Yaskawa INFORM job: X2_8A-21A(90,0)_REV_O.JBI

/JOB
//NAME X2_8A-21A(90,0)_REV_O
///FOLDERNAME X2
//POS
///NPOS 1933,1933,1933,50,0,0
///TOOL 0
///POSTYPE PULSE
///PULSE
C00000=-12667,-135547,-130714,31270,45596,0
C00001=-9315,-159766,-119262,-3212,6219,55552
C00002=-157761,-135547,-130714,31270,45596,-69143
C00003=-154472,-113934,-104337,41712,51336,-70449
C00004=-149832,-108771,-100172,39130,49259,-68869
C00005=-148058,-106656,-98467,38074,48499,-68236
C00006=-148062,-106275,-96666,38578,47777,-68578
C00007=-148058,-106656,-98467,38074,48499,-68236
C00008=-147997,-106381,-96958,38469,47847,-68508
C00009=-145894,-104035,-96109,36815,47477,-67498
C00010=-147997,-106381,-96958,38469,47847,-68508
C00011=-154410,-113635,-102825,42095,50721,-70729
C00012=-154342,-120637,-107041,25827,48602,-38771
C00013=-150292,-111683,-102360,22573,48994,-36710
C00014=-148798,-108210,-100464,21373,49171,-35962
C00015=-146664,-105787,-99597,19708,49308,-34937
C00016=-146949,-106220,-99797,19932,49282,-35074
C00017=-147721,-103636,-97533,20478,49410,-35405
C00018=-146949,-106220,-99797,19932,49282,-35074
C00019=-152261,-118724,-106469,24248,48548,-37770
C00020=-148295,-114597,-117137,-6490,60568,-69086
C00021=-147868,-109631,-111600,-6790,59752,-68875
C00022=-117093,-120499,-115228,-23648,62285,-57221
C00023=-113886,-102168,-107256,-24278,67338,-57062
C00024=-113886,-102375,-106001,-24426,66534,-56885
C00025=-113886,-102359,-106115,-24413,66607,-56901
C00026=-113886,-102359,-106115,-24413,66607,-56901
C00027=-114646,-97769,-104385,-23859,67577,-57404
C00028=-114475,-101992,-107821,-23944,67574,-57337
C00029=-147704,-107727,-109395,-6911,59390,-68790
C00030=-147708,-107860,-107783,-6984,58336,-68724
C00031=-147704,-107727,-109395,-6911,59390,-68790
C00032=-147723,-107760,-107968,-6963,58499,-68740
C00033=-147306,-102596,-106094,-7098,60024,-68678
C00034=-147723,-107760,-107968,-6963,58499,-68740
C00035=-148315,-114751,-115749,-6537,59639,-69038
C00036=-148355,-114889,-117236,-6461,60467,-69101
C00037=-147925,-109892,-111692,-6763,59663,-68890
C00038=-147761,-107977,-109485,-6884,59305,-68805
C00039=-147764,-108104,-107870,-6957,58254,-68739
C00040=-147777,-108153,-108078,-6942,58354,-68751
C00041=-147358,-102980,-106206,-7078,59886,-68688
C00042=-147777,-108153,-108078,-6942,58354,-68751
C00043=-148373,-115211,-115873,-6515,59468,-69049
C00044=-147696,-122269,-111871,-35505,39043,-51945
C00045=-147690,-118447,-100224,-39719,34874,-49579
C00046=-148491,-109409,-94254,-38171,35277,-50420
C00047=-148787,-105724,-91002,-38010,35060,-50504
C00048=-148789,-105382,-89977,-38411,34697,-50285
C00049=-149058,-101689,-89016,-37046,35623,-51030
C00050=-149145,-100783,-88679,-36755,35795,-51189
C00051=-149058,-101689,-89016,-37046,35623,-51030
C00052=-145777,-99657,-88811,-39022,37803,-49998
C00053=-148139,-100407,-89095,-37251,36591,-50936
C00054=-145777,-99657,-88811,-39022,37803,-49998
C00055=-147690,-118447,-100224,-39719,34874,-49579
C00056=-128033,-128545,-103748,-39689,32513,-43973
C00057=-128383,-118409,-97778,-37905,33566,-44930
C00058=-128511,-114277,-94563,-37658,33626,-45064
C00059=-128512,-113804,-93446,-38069,33271,-44843
C00060=-129119,-111006,-93029,-36452,33958,-45715
C00061=-129434,-109852,-92636,-35862,34111,-46033
C00062=-128358,-113721,-93936,-37885,33613,-44941
C00063=-176216,-70111,-78093,55162,70856,-80763
C00064=-174311,-70781,-78417,54616,69674,-80426
C00065=-176216,-70111,-78093,55162,70856,-80763
C00066=-181747,-69996,-81392,56304,75271,-81045
C00067=-178033,-77165,-93769,42680,75059,-77098
C00068=-164745,-109340,-116699,-3009,62053,-68278
C00069=-145851,-112599,-102075,-47717,41998,-56322
C00070=-148044,-104803,-96379,-45883,41204,-57334
C00071=-148864,-101708,-93474,-45490,40644,-57533
C00072=-148866,-101457,-92299,-45986,40221,-57239
C00073=-148863,-101834,-94104,-45225,40876,-57690
C00074=-145127,-99228,-91361,-47944,42572,-56214
C00075=-147466,-100038,-91670,-46636,41186,-56907
C00076=-145127,-99228,-91361,-47944,42572,-56214
C00077=-146129,-107372,-95667,-48598,40993,-55782
C00078=-148216,-109089,-93488,-49289,38371,-55335
C00079=-148344,-107837,-93052,-48851,38553,-55585
C00080=-147906,-112054,-94498,-50363,37947,-54724
C00081=-145851,-112599,-102075,-47717,41998,-56322
C00082=-158250,-140903,-124067,-47621,67451,-49320
C00083=-161740,-133075,-117656,-46661,65672,-50232
C00084=-162335,-130592,-114553,-46699,64919,-50156
C00085=-162276,-129951,-113381,-46845,64676,-49998
C00086=-160420,-132544,-115533,-47350,65644,-49520
C00087=-135901,-74424,-73697,-74364,100921,-31256
C00088=-137788,-75503,-74147,-74218,99532,-31324
C00089=-138769,-76027,-74362,-74146,98812,-31363
C00090=-135901,-74424,-73697,-74364,100921,-31256
C00091=-149282,-147643,-98518,-79858,51263,-26133
C00092=-149394,-146891,-98381,-79629,51249,-26315
C00093=-148448,-152811,-99407,-81432,51428,-24854
C00094=-139735,-166147,-105854,-82069,56849,-22658
C00095=-180438,-97574,-115199,-33764,102267,52414
C00096=-189965,-108899,-115705,-31971,94091,51156
C00097=-190633,-110068,-115194,-31831,93066,51189
C00098=-190637,-110288,-114404,-31804,92551,51332
C00099=-190629,-109833,-115910,-31859,93547,51055
C00100=-186867,-102382,-113240,-32521,96788,51574
C00101=-187005,-102964,-110979,-32373,95300,51952
C00102=-188888,-106610,-112304,-32065,93703,51681
C00103=-187005,-102964,-110979,-32373,95300,51952
C00104=-188021,-107681,-112675,-32159,93748,52003
C00105=-189590,-103281,-111094,-32025,94271,51250
C00106=-188021,-107681,-112675,-32159,93748,52003
C00107=-180438,-97574,-115199,-33764,102267,52414
C00108=-185735,-83978,-109774,-33564,103394,50026
C00109=-199988,-77820,-108712,11582,98175,-38155
C00110=-204749,-56978,-92496,29836,109182,-47433
C00111=-202460,-56662,-91339,29422,107990,-46925
C00112=-201413,-57385,-91726,29256,107546,-46663
C00113=-201611,-57041,-91542,29296,107663,-46703
C00114=-201611,-58240,-90431,29070,106521,-47008
C00115=-203359,-50274,-87822,29763,109247,-46906
C00116=-195470,-25798,-72981,29209,109868,-43903
C00117=-195013,-27562,-73704,29036,109327,-43888
C00118=-194283,-28250,-74172,28893,109053,-43704
C00119=-194480,-28066,-74047,28932,109127,-43754
C00120=-194480,-29296,-73135,28708,108075,-44034
C00121=-195605,-24849,-71507,29147,109538,-44038
C00122=-191110,-5546,-57842,28597,109561,-42465
C00123=-192519,-3768,-54500,33008,111368,-41387
C00124=-191992,-5303,-55742,32912,111174,-41254
C00125=-192059,-5108,-55586,32924,111198,-41271
C00126=-192059,-6294,-54683,32651,110210,-41583
C00127=-192882,-2296,-53893,33162,111810,-41382
C00128=-203365,-15491,-64400,34648,115083,-44256
C00129=-218411,-26661,-75493,58573,107247,-46176
C00130=-145332,-87800,-123084,4045,108310,15756
C00131=-109199,-104290,-129101,-21867,105305,43874
C00132=-112610,-115777,-129409,-14908,94573,36374
C00133=-117115,-112620,-124614,-14006,92529,35127
C00134=-122920,-112365,-123082,-12804,90828,33394
C00135=-122920,-112757,-122533,-12801,90299,33450
C00136=-122920,-112643,-122701,-12801,90458,33434
C00137=-123525,-106184,-120478,-12700,92275,33049
C00138=-122920,-112643,-122701,-12801,90458,33434
C00139=-99736,-107822,-114568,-33675,94477,38345
C00140=-104025,-110392,-115465,-33031,92199,37352
C00141=-122920,-112281,-123196,-12806,90936,33384
C00142=-119624,-116552,-128230,-13509,92325,34321
C00143=-118894,-118314,-126738,-16484,89836,32308
C00144=-120722,-107922,-120892,-16116,91165,31519
C00145=-120722,-108682,-119869,-16105,90184,31649
C00146=-120722,-108549,-120061,-16106,90363,31625
C00147=-121452,-100742,-117219,-15984,92406,31115
C00148=-121469,-105211,-119242,-15960,91389,31241
C00149=-101189,-106149,-119574,-19874,95347,37480
C00150=-117231,-121833,-124467,-22052,85463,28755
C00151=-122341,-114124,-118662,-20866,84531,27121
C00152=-123318,-113111,-117155,-20643,83910,26885
C00153=-123641,-113323,-116249,-20585,83205,26892
C00154=-123595,-112804,-116375,-20585,83540,26851
C00155=-123397,-106736,-114247,-20589,85286,26623
C00156=-123595,-112804,-116375,-20585,83540,26851
C00157=-116023,-114044,-115764,-22346,84523,29358
C00158=-117346,-116777,-115957,-22098,82979,29171
C00159=-118867,-116723,-116143,-21757,82713,28674
C00160=-116293,-116772,-115815,-22329,83179,29512
C00161=-117231,-121833,-124467,-22052,85463,28755
C00162=-154726,-134692,-133300,19029,79240,32627
C00163=-155157,-123239,-125350,19102,80279,32639
C00164=-157379,-119183,-122744,19707,81244,32017
C00165=-157379,-119362,-122195,19727,80834,31951
C00166=-157379,-119302,-122385,19720,80973,31974
C00167=-156300,-113680,-120537,19346,82380,32578
C00168=-157190,-118033,-122826,19626,81802,32175
C00169=-175737,-146891,-124533,43519,91428,21152
C00170=-174721,-145732,-123510,43532,90901,21397
C00171=-174058,-146263,-122600,43517,89962,21303
C00172=-174118,-146172,-122608,43517,90030,21304
C00173=-173980,-142501,-121319,43546,90763,21685
C00174=-177980,-148291,-122807,43386,91220,20037
C00175=-177422,-148804,-122388,43393,90560,20012
C00176=-177529,-148647,-122416,43390,90685,20016
C00177=-177298,-142861,-120187,43458,91752,20577
C00178=-177298,-144596,-123184,43505,92454,20876
C00179=-171479,-146654,-130538,32727,84182,23892
C00180=-166226,-153583,-132379,32233,80103,24817
C00181=-165373,-149023,-130107,32047,80585,25297
C00182=-165373,-148396,-128971,32075,80265,25206
C00183=-165373,-148499,-129154,32071,80317,25220
C00184=-163349,-139759,-126762,31573,82140,26540
C00185=-164602,-145870,-129723,31842,81480,25858
C00186=-94432,-122903,-125032,-9527,78085,47389
C00187=-94433,-123258,-123690,-9573,77094,47468
C00188=-95155,-123271,-123048,-9356,76614,47257
C00189=-95046,-123163,-123057,-9388,76686,47288
C00190=-95200,-117884,-121168,-9287,78202,47121
C00191=-91884,-123031,-122816,-10395,76986,48348
C00192=-93089,-124364,-122323,-10053,75863,48028
C00193=-92985,-124257,-122339,-10083,75941,48058
C00194=-93121,-120077,-120785,-9995,77098,47917
C00195=-92614,-123227,-123779,-10148,77379,48067
C00196=-142492,-148036,-131704,16940,70784,31434
C00197=-120610,-122471,-119242,-21572,81234,22537
C00198=-120610,-122484,-118172,-21604,80613,22649
C00199=-120610,-122391,-116483,-21658,79689,22817
C00200=-120610,-122419,-116833,-21647,79876,22783
C00201=-120610,-122423,-116832,-21647,79874,22783
C00202=-120610,-122419,-116833,-21647,79876,22783
C00203=-120610,-122416,-116761,-21649,79836,22790
C00204=-120610,-122436,-116768,-21650,79830,22791
C00205=-120610,-122416,-116761,-21649,79836,22790
C00206=-120611,-122370,-120508,-21535,82009,22397
C00207=-120500,-119354,-126515,-17332,87675,17755
C00208=-155157,-123239,-125350,19102,80279,32639
C00209=-157379,-119183,-122744,19707,81244,32017
C00210=-157379,-119362,-122195,19727,80834,31951
C00211=-157379,-119302,-122385,19720,80973,31974
C00212=-156300,-113680,-120537,19346,82380,32578
C00213=-157190,-118033,-122826,19626,81802,32175
C00214=-175737,-146891,-124533,43519,91428,21152
C00215=-174721,-145732,-123510,43532,90901,21397
C00216=-174058,-146263,-122600,43517,89962,21303
C00217=-174118,-146172,-122608,43517,90030,21304
C00218=-173980,-142501,-121319,43546,90763,21685
C00219=-177980,-148291,-122807,43386,91220,20037
C00220=-177422,-148804,-122388,43393,90560,20012
C00221=-177529,-148647,-122416,43390,90685,20016
C00222=-177298,-142861,-120187,43458,91752,20577
C00223=-177298,-144596,-123184,43505,92454,20876
C00224=-171479,-146654,-130538,32727,84182,23892
C00225=-166226,-153583,-132379,32233,80103,24817
C00226=-165373,-149023,-130107,32047,80585,25297
C00227=-165373,-148396,-128971,32075,80265,25206
C00228=-165373,-148499,-129154,32071,80317,25220
C00229=-163349,-139759,-126762,31573,82140,26540
C00230=-164602,-145870,-129723,31842,81480,25858
C00231=-94432,-122903,-125032,-9527,78085,47389
C00232=-94433,-123258,-123690,-9573,77094,47468
C00233=-95155,-123271,-123048,-9356,76614,47257
C00234=-95046,-123163,-123057,-9388,76686,47288
C00235=-95200,-117884,-121168,-9287,78202,47121
C00236=-91884,-123031,-122816,-10395,76986,48348
C00237=-93089,-124364,-122323,-10053,75863,48028
C00238=-92985,-124257,-122339,-10083,75941,48058
C00239=-93121,-120077,-120785,-9995,77098,47917
C00240=-92614,-123227,-123779,-10148,77379,48067
C00241=-120611,-118687,-129075,-3134,90000,4412
C00242=-148570,-103220,-123870,3202,94742,-4439
C00243=-148570,-107981,-119269,3182,89471,-4572
C00244=-127056,-134876,-126643,7466,81568,-11458
C00245=-127056,-134636,-125176,7474,80796,-11503
C00246=-127056,-134735,-125722,7473,81078,-11487
C00247=-126802,-126383,-123229,7383,83789,-11239
C00248=-127056,-134735,-125722,7473,81078,-11487
C00249=-152011,-114496,-114941,26277,90880,-36116
C00250=-148601,-117726,-116011,25806,88925,-35294
C00251=-149160,-116575,-119890,25935,91789,-34871
C00252=-149049,-114583,-124201,25964,95071,-34011
C00253=-120621,-113915,-131911,-13153,116790,34478
C00254=-136832,-143297,-133894,-19017,104291,40845
C00255=-187686,-122249,-118318,-34521,102174,42234
C00256=-187703,-122088,-115580,-34298,100833,42653
C00257=-187707,-122010,-114917,-34250,100525,42749
C00258=-187713,-121734,-113169,-34135,99743,42991
C00259=-187707,-122010,-114917,-34250,100525,42749
C00260=-187770,-121697,-112491,-32279,113674,44764
C00261=-187767,-121692,-112491,-32279,113678,44765
C00262=-187770,-121697,-112491,-32279,113674,44764
C00263=-187667,-121438,-112064,-34928,84963,41689
C00264=-187673,-121448,-112068,-34927,84958,41688
C00265=-187667,-121438,-112064,-34928,84963,41689
C00266=-187641,-121360,-124129,-34919,91154,39753
C00267=-178673,-119471,-127738,-23493,103847,53429
C00268=-198679,-138959,-135715,-16358,95506,85843
C00269=-190587,-123959,-122502,-31374,99801,86508
C00270=-192699,-142870,-125546,-30768,92257,87745
C00271=-192699,-141891,-123487,-30748,91600,87922
C00272=-192699,-142870,-125546,-30768,92257,87745
C00273=-239187,-117092,-121328,-77,117937,72244
C00274=-239070,-127403,-124585,-50,114644,72291
C00275=-197002,-104016,-110014,-22827,126025,83305
C00276=-198918,-110501,-112317,-22907,123733,82993
C00277=-197002,-103017,-112874,-23585,128123,82776
C00278=-191212,-108340,-120713,-19480,129464,82344
C00279=-160879,-120821,-131564,-37,121469,81968
C00280=-157394,-128671,-131753,738,117538,83283
C00281=-158801,-138021,-132727,409,113343,82737
C00282=-158801,-138035,-132347,409,113101,82737
C00283=-158801,-138034,-131509,408,112586,82736
C00284=-158801,-138039,-131833,408,112783,82736
C00285=-160693,-149427,-134985,6,108877,82039
C00286=-160612,-153549,-136083,24,107435,82069
C00287=-159125,-144348,-133603,336,110634,82611
C00288=-199963,-104116,-119881,11013,127404,83152
C00289=-204692,-116225,-118816,8637,121169,80600
C00290=-203581,-121519,-120530,8810,119404,80895
C00291=-204849,-113790,-122122,8953,124435,80816
C00292=-166129,-114439,-129167,13521,133132,-54375
C00293=-82387,-124374,-130385,21792,102809,-55833
C00294=-37550,-124758,-124791,27166,84975,-54517
C00295=-35933,-124831,-122904,26864,83389,-54284
C00296=-35589,-124875,-121597,26827,82538,-54351
C00297=-35584,-124889,-121174,26839,82296,-54405
C00298=-35764,-126387,-121953,26892,82093,-54519
C00299=-31633,-125451,-121673,25972,81076,-53208
C00300=-35764,-126387,-121953,26892,82093,-54519
C00301=-46981,-157328,-126723,35790,81436,-33730
C00302=-42905,-153934,-122174,35701,78867,-32870
C00303=-42758,-143813,-119569,35389,81762,-31868
C00304=-42905,-153934,-122174,35701,78867,-32870
C00305=-53188,-117519,-120731,36414,97747,-30962
C00306=-95179,-109851,-129540,3422,106316,17944
C00307=-143691,-100776,-119079,-26047,122130,73021
C00308=-146029,-112499,-120098,-24937,116556,73463
C00309=-147204,-116618,-119576,-24569,113992,73590
C00310=-147487,-116577,-118677,-24502,113425,73607
C00311=-146967,-116625,-120319,-24630,114475,73574
C00312=-147345,-121113,-121824,-24401,113105,73737
C00313=-146899,-128254,-123879,-23878,111030,74376
C00314=-147345,-121113,-121824,-24401,113105,73737
C00315=-118081,-135478,-120686,-30293,109901,65237
C00316=-118366,-136707,-118609,-29972,108136,65614
C00317=-120887,-140213,-119894,-30302,106351,65070
C00318=-118366,-136707,-118609,-29972,108136,65614
C00319=-117820,-130449,-123242,-31209,113594,64262
C00320=-143015,-142486,-131518,-29087,102599,89323
C00321=-146039,-130109,-126790,-30266,105409,87337
C00322=-146039,-130165,-125281,-30113,104578,87565
C00323=-146020,-130184,-125355,-30122,104615,87562
C00324=-146020,-130184,-125484,-30134,104685,87544
C00325=-147293,-140381,-128439,-29740,101251,87961
C00326=-146475,-133913,-127536,-30061,103955,87559
C00327=-159288,-132688,-127179,-30476,99746,83631
C00328=-162405,-133989,-127560,-30412,98256,82812
C00329=-162405,-133889,-126354,-30348,97657,82974
C00330=-162405,-133904,-126492,-30355,97724,82955
C00331=-162405,-133904,-126492,-30355,97724,82955
C00332=-164001,-141203,-128579,-30154,95010,83056
C00333=-163239,-137919,-128550,-30280,96734,82895
C00334=-145009,-133074,-127629,-29362,102627,83449
C00335=-93926,-103398,-125362,-18301,106221,39936
C00336=-72688,-110808,-124077,-7134,85250,24096
C00337=-72688,-113152,-120783,-7167,82043,24279
C00338=-76579,-98113,-113117,-5975,84731,22871
C00339=-76579,-98978,-111730,-5983,83442,22935
C00340=-76579,-98797,-112043,-5982,83725,22921
C00341=-78138,-93000,-109805,-5503,85212,22351
C00342=-76410,-98400,-113840,-6024,85039,22913
C00343=-76410,-94572,-117616,-6016,89307,22709
C00344=-77214,-94325,-113861,-5779,87079,22562
C00345=-77214,-95141,-112958,-5781,86109,22607
C00346=-77214,-94950,-113181,-5780,86344,22597
C00347=-78619,-89504,-111030,-5355,87721,22093
C00348=-77257,-93804,-114159,-5765,87526,22530
C00349=-83348,-134113,-127593,-4031,74771,21021
C00350=-84698,-126818,-124628,-3579,76630,20501
C00351=-84698,-126887,-123754,-3584,76055,20517
C00352=-84698,-126872,-123997,-3581,76213,20513
C00353=-86532,-116989,-120868,-2976,79288,19814
C00354=-85417,-122616,-124575,-3327,78721,20200
C00355=-140085,-104632,-109249,40944,98797,-6712
C00356=-140263,-103640,-106572,40817,98007,-7102
C00357=-138995,-104322,-106820,40710,97277,-6835
C00358=-140263,-103640,-106572,40817,98007,-7102
C00359=-135988,-101428,-112112,41019,99549,-4631
C00360=-141957,-83285,-117139,12315,91699,6710
C00361=-161957,-129781,-122866,-20018,67926,12328
C00362=-166016,-109699,-113650,-17211,72980,10098
C00363=-166795,-105246,-111748,-16434,74862,9605
C00364=-165677,-113012,-111900,-18316,68836,10778
C00365=-162725,-116093,-113629,-19548,69016,11850
C00366=-162651,-107484,-110669,-19284,71494,11460
C00367=-162725,-116093,-113629,-19548,69016,11850
C00368=-155151,-112727,-112486,-22270,71877,14160
C00369=-155120,-113819,-110277,-22518,70103,14518
C00370=-159000,-114269,-110433,-21107,68960,13264
C00371=-155120,-113819,-110277,-22518,70103,14518
C00372=-155137,-138999,-124748,-23105,66364,15269
C00373=-81055,-115973,-127517,23586,109336,-64560
C00374=-76492,-127739,-126040,22738,101683,-64421
C00375=-76072,-128597,-125529,22671,100870,-64425
C00376=-76065,-128640,-125326,22657,100732,-64448
C00377=-76072,-128576,-125785,22685,101025,-64394
C00378=-82641,-146978,-130130,22016,96499,-67668
C00379=-81130,-155003,-132256,21951,93476,-67670
C00380=-82641,-146978,-130130,22016,96499,-67668
C00381=-84000,-144678,-127518,21929,96467,-68175
C00382=-84000,-143983,-126065,21900,95967,-68269
C00383=-83327,-146231,-127404,21916,95478,-68108
C00384=-88356,-135439,-132684,22407,104994,-68175
C00385=-104080,-128245,-132212,-31995,84146,-22143
C00386=-106783,-105266,-117364,-31197,85468,-23533
C00387=-107129,-103609,-115494,-31111,85090,-23558
C00388=-107127,-104217,-114421,-31144,84251,-23329
C00389=-107044,-104571,-114816,-31164,84333,-23320
C00390=-107880,-99055,-112779,-30885,85404,-23924
C00391=-107044,-104571,-114816,-31164,84333,-23320
C00392=-105114,-115284,-123193,-31689,84721,-22698
C00393=-105208,-113465,-123990,-31624,85910,-23065
C00394=-106823,-104635,-117017,-31184,85549,-23570
C00395=-107122,-103295,-115264,-31113,85109,-23561
C00396=-107121,-103855,-114286,-31142,84342,-23351
C00397=-107087,-104437,-114776,-31151,84356,-23343
C00398=-107921,-98925,-112738,-30873,85426,-23945
C00399=-107087,-104437,-114776,-31151,84356,-23343
C00400=-105701,-116384,-125830,-31502,85418,-23114
C00401=-63541,-120749,-127234,-38861,101172,-11499
C00402=-62914,-102725,-115578,-39257,103083,-11954
C00403=-62914,-103574,-114098,-39030,102025,-11552
C00404=-62914,-103512,-114221,-39048,102111,-11585
C00405=-65395,-98857,-112499,-39034,102095,-12627
C00406=-63190,-103387,-116908,-39318,103341,-12168
C00407=-105701,-116384,-125830,-31502,85418,-23114
C00408=-79137,-116524,-127291,-7118,77084,38210
C00409=-66518,-158449,-133200,-8588,59166,50817
C00410=-70166,-147728,-127011,-6864,60501,49298
C00411=-71549,-143558,-123868,-6244,60595,48757
C00412=-71544,-142942,-122687,-6271,60188,48782
C00413=-71412,-140542,-122600,-6259,61371,48766
C00414=-74130,-137647,-121783,-5023,62161,47690
C00415=-71412,-140542,-122600,-6259,61371,48766
C00416=-59221,-85077,-106862,-19044,97138,55247
C00417=-59772,-90133,-108950,-18878,95774,55276
C00418=-59221,-85077,-106862,-19044,97138,55247
C00419=-65406,-128676,-128270,-8670,80773,42177
C00420=-57064,-112054,-129147,-2862,108793,29097
C00421=-70948,-123089,-127271,10962,111372,-380
C00422=-67644,-116564,-123033,11394,111660,848
C00423=-67644,-116773,-122597,11361,111292,811
C00424=-67644,-116291,-123546,11437,112109,893
C00425=-70770,-123262,-125779,10903,110357,-412
C00426=-70770,-123588,-124717,10837,109552,-488
C00427=-69306,-120453,-123728,11077,110342,115
C00428=-70770,-123283,-125719,10898,110311,-416
C00429=-70770,-119886,-130778,11344,115083,53
C00430=-68413,-122856,-123349,22437,117236,58
C00431=-67404,-122631,-120786,22344,115611,123
C00432=-67401,-122683,-120099,22253,115193,37
C00433=-67283,-122594,-120333,22317,115338,115
C00434=-65261,-118175,-118917,23034,116088,1096
C00435=-67283,-122594,-120333,22317,115338,115
C00436=-70820,-123560,-126018,22187,119059,-540
C00437=-59587,-128850,-129971,-18356,103459,48793
C00438=-60648,-112549,-116046,-37363,97913,74718
C00439=-66648,-121539,-115269,-36526,91263,74498
C00440=-69624,-125916,-115212,-36242,88151,74300
C00441=-69624,-125773,-114639,-36242,87924,74374
C00442=-69624,-125814,-114800,-36242,87987,74354
C00443=-70738,-127677,-115368,-36152,87024,74211
C00444=-69624,-125814,-114800,-36242,87987,74354
C00445=-61556,-115340,-115782,-37136,96245,74919
C00446=-93863,-107857,-129738,-18786,98098,27923
C00447=-113340,-105978,-120535,-17383,92037,15860
C00448=-116256,-99504,-115214,-16745,91512,14962
C00449=-117355,-97038,-113094,-16498,91266,14630
C00450=-124053,-106600,-116618,-14934,87391,12894
C00451=-123019,-109757,-118902,-15179,87365,13243
C00452=-120254,-118381,-124729,-15823,87055,14212
C00453=-121076,-118719,-112405,-41381,81563,9211
C00454=-125328,-110839,-107644,-40465,80446,7775
C00455=-126920,-107772,-105722,-40091,80023,7243
C00456=-122279,-105715,-102241,-45382,81605,7865
C00457=-118123,-103314,-98388,-50429,83325,8212
C00458=-115452,-99808,-95169,-50805,84680,8860
C00459=-113598,-101964,-96694,-51043,85596,9323
C00460=-108732,-107177,-100380,-51565,88044,10518
C00461=-131658,-113091,-133069,-11905,90618,-13395
C00462=-155934,-143784,-122811,23124,58745,-32427
C00463=-151507,-132468,-117411,20635,59886,-30339
C00464=-149876,-128251,-115276,19729,60288,-29596
C00465=-151213,-128323,-114307,20456,60014,-30191
C00466=-146890,-120795,-114089,13688,65901,-25886
C00467=-142734,-111238,-112703,7950,73001,-22079
C00468=-143750,-114926,-115045,8343,72653,-22456
C00469=-146492,-125018,-121022,9420,71459,-23506
C00470=-146459,-122334,-129315,9145,77857,-23007
C00471=-118526,-115013,-133262,8809,105739,-46794
C00472=-93674,-118800,-129721,8134,120991,-68616
C00473=-93669,-120967,-127104,7892,118292,-68817
C00474=-94465,-127736,-127937,7493,115415,-69310
C00475=-101667,-152205,-134731,5550,107657,-72408
C00476=-93660,-121042,-127131,7893,118270,-68815
C00477=-93665,-118880,-129750,8134,120967,-68614
C00478=-98446,-113408,-116165,41475,93741,-73013
C00479=-95217,-118830,-115137,40946,89638,-73223
C00480=-92806,-121560,-115150,40665,87459,-73017
C00481=-95954,-130241,-115077,41081,85472,-75169
C00482=-96936,-125131,-114749,41104,87782,-74702
C00483=-101504,-121000,-116278,41571,92256,-74948
C00484=-100864,-122088,-112493,43204,76282,-71688
C00485=-96953,-122826,-110054,42689,72984,-71279
C00486=-94247,-124338,-109802,42269,70974,-70864
C00487=-94193,-123974,-108080,42453,70297,-71131
C00488=-95642,-121622,-108630,42447,72155,-71017
C00489=-100864,-121830,-111367,43291,75868,-71867
C00490=-131033,-115476,-133015,2815,101744,-74384
C00491=-151471,-119125,-123137,-34971,103386,-73225
C00492=-162012,-101235,-114016,-37763,108592,-75954
C00493=-165297,-105997,-114400,-37202,105452,-76208
C00494=-161279,-107047,-112450,-36906,105725,-74600
C00495=-157962,-101866,-111865,-37402,108959,-74341
C00496=-155898,-93647,-112180,-38609,113341,-75115
C00497=-93674,-112333,-133466,8753,126560,-68151
C00498=-93674,-118800,-129721,8134,120991,-68616
C00499=-93669,-120967,-127104,7892,118292,-68817
C00500=-93667,-121558,-126026,7814,117333,-68886
C00501=-93663,-121536,-126144,7822,117416,-68879
C00502=-93639,-121762,-126135,7818,117296,-68878
C00503=-93680,-121434,-126040,7817,117406,-68885
C00504=-93660,-121042,-127131,7893,118270,-68815
C00505=-93665,-118880,-129750,8134,120967,-68614
C00506=-98446,-113408,-116165,41475,93741,-73013
C00507=-93996,-117843,-114815,40802,89312,-72817
C00508=-91343,-117266,-113836,40455,87860,-72224
C00509=-92137,-119395,-114109,40564,87510,-72703
C00510=-95072,-126184,-113786,40951,86041,-74561
C00511=-95071,-125918,-112907,40977,85731,-74679
C00512=-96936,-125131,-114749,41104,87782,-74702
C00513=-101504,-121000,-116278,41571,92256,-74948
C00514=-100864,-122088,-112493,43204,76282,-71688
C00515=-95643,-121963,-109784,42340,72556,-70846
C00516=-93677,-120964,-108398,41948,71358,-70433
C00517=-93599,-120925,-107098,42100,70733,-70661
C00518=-95642,-121622,-108630,42447,72155,-71017
C00519=-100864,-121830,-111367,43291,75868,-71867
C00520=-131033,-115476,-133015,2815,101744,-74384
C00521=-151471,-119125,-123137,-34971,103386,-73225
C00522=-162012,-101235,-114016,-37763,108592,-75954
C00523=-163593,-104354,-113811,-37340,106547,-75879
C00524=-162938,-104376,-113793,-37349,106803,-75692
C00525=-158829,-104862,-111593,-37019,107224,-74083
C00526=-157962,-101866,-111865,-37402,108959,-74341
C00527=-155898,-93647,-112180,-38609,113341,-75115
C00528=-179206,-139250,-107986,-62075,77828,-66561
C00529=-185232,-138953,-105140,-62379,73225,-66913
C00530=-187696,-139015,-104542,-62453,71468,-67163
C00531=-187702,-137665,-102648,-62587,71237,-66963
C00532=-185238,-138055,-103864,-62461,73065,-66778
C00533=-179211,-138396,-106727,-62132,77661,-66424
C00534=-179188,-148562,-121526,-61524,79591,-68010
C00535=-184417,-115822,-131978,-19629,107310,7500
C00536=-190427,-134899,-136820,8574,116374,78562
C00537=-186100,-113471,-128285,10018,121587,80668
C00538=-191225,-146270,-136079,6950,104131,75337
C00539=-190490,-140209,-134074,7301,107114,76191
C00540=-191198,-135798,-132689,7359,109020,76211
C00541=-188542,-139162,-133652,7636,107649,77074
C00542=-188892,-120096,-126431,8986,117412,79228
C00543=-186988,-122354,-127008,9286,116409,79864
C00544=-188900,-120476,-124632,-3181,115072,77765
C00545=-188087,-121040,-124812,-3025,114921,78067
C00546=-187942,-121398,-126015,-3016,115485,78109
C00547=-187937,-119495,-128851,-3098,118205,78035
C00548=-176042,-128909,-129640,-7380,110692,58022
C00549=-187833,-113452,-115854,-34994,105139,41767
C00550=-187847,-113781,-113588,-34722,103839,42187
C00551=-187853,-113844,-112659,-34623,103335,42348
C00552=-187856,-113866,-111596,-34519,102780,42525
C00553=-187851,-113844,-112538,-34611,103274,42368
C00554=-187836,-113627,-114840,-34866,104547,41960
C00555=-186756,-108501,-120882,-36201,110201,40487
C00556=-150585,-129060,-123753,-46684,114085,-39870
C00557=-134046,-137019,-115206,-49635,112096,-74674
C00558=-134033,-140586,-110307,-48065,108843,-72866
C00559=-134037,-138671,-107458,-47843,108316,-72589
C00560=-133950,-137111,-106105,-47812,108341,-72556
C00561=-134016,-151531,-126358,1136,113524,-57559
C00562=-134135,-151353,-126308,1093,113591,-57603
C00563=-135498,-150804,-126324,2361,113462,-57532
C00564=-137673,-151162,-132623,1623,117206,-58299
C00565=-106012,-107394,-121753,14018,130776,-44816
C00566=-106669,-102485,-112824,13121,127987,-45519
C00567=-97512,-96218,-110425,14566,129183,-82759
C00568=-98864,-105619,-112306,13303,125832,-83842
C00569=-106150,-109468,-113796,12766,125107,-45727
C00570=-105474,-116823,-114648,29161,97726,-33837
C00571=-134074,-146851,-118858,40485,90771,-46834
C00572=-138964,-153067,-136534,10460,111077,-51089
C00573=-145533,-126220,-133766,11748,110749,-32017
C00574=-159341,-97264,-124494,3811,101460,647
C00575=-162841,-115960,-130919,4373,95984,-637
C00576=-188071,-112180,-99768,1790,31671,46486
C00577=-188092,-111455,-97340,1875,30550,46442
C00578=-187851,-111485,-96835,1581,30220,46589
C00579=-187792,-110201,-93997,1555,29133,46605
C00580=-187737,-110060,-93474,1490,28882,46636
C00581=-187785,-109075,-90961,1604,27844,46576
C00582=-188106,-109627,-92159,2030,28303,46362
C00583=-188086,-110531,-94662,1935,29378,46411
C00584=-188086,-114129,-114927,1479,39995,46659
C00585=-201470,-41376,-102585,19941,97743,-57993
C00586=-197439,-2624,-49840,39121,107911,-51008
C00587=-168348,92819,48556,27514,116832,-48709
C00588=-170146,82769,36005,28011,119675,-48673
C00589=-172466,59662,8523,30747,114377,-38085
C00590=-173361,44293,-8668,31536,116980,-37634
C00591=-173326,42548,-10417,31798,119739,-39927
C00592=-173293,31446,-22173,31559,124382,-42741
C00593=-170045,43132,-9775,28753,130915,-51393
C00594=-186843,33187,-28183,45340,118495,-56566
C00595=-187270,22965,-40018,42118,113549,-44205
C00596=-164927,12374,-50848,37497,97302,26684
C00597=-160848,-52651,-98971,6904,73590,44156
C00598=-187933,-111679,-98706,-278,30585,46526
C00599=-187953,-110958,-96368,-260,29517,46517
C00600=-188171,-110591,-95666,34,29272,46369
C00601=-188111,-109885,-93130,-50,28074,46412
C00602=-188090,-109778,-92606,-82,27808,46427
C00603=-188055,-108797,-90194,-133,26826,46455
C00604=-187968,-109087,-91174,-258,27282,46516
C00605=-187948,-109974,-93584,-278,28309,46526
C00606=-190713,-138118,-122139,3147,45685,54861
C00607=-188097,-104568,-127563,3199,90457,72619
C00608=-188112,-108983,-124849,3203,86524,72515
C00609=-196049,-130715,-128058,11352,73875,69900
C00610=-196049,-130372,-129815,11289,75109,70015
C00611=-199069,-128516,-127529,12349,75098,68966
C00612=-193131,-119078,-125609,7963,80164,71095
C00613=-187481,-125068,-127230,2773,76551,72417
C00614=-191681,-130682,-128318,6769,73360,71103
C00615=-188153,-109076,-124888,3215,86502,72501
C00616=-188138,-104664,-127604,3212,90434,72606
C00617=-187898,-111965,-120493,-16766,69565,69566
C00618=-187918,-113285,-117348,-17044,67055,69927
C00619=-188433,-114855,-116277,-16981,65546,69965
C00620=-188279,-112660,-115510,-16972,66207,69918
C00621=-188300,-112703,-115461,-16971,66156,69920
C00622=-188153,-111836,-115149,-17009,66426,69933
C00623=-187944,-113344,-117352,-17035,67023,69922
C00624=-187924,-112030,-120500,-16757,69531,69561
C00625=-180038,-109975,-126789,-2440,82512,-7441
C00626=-174468,-102021,-118148,-1871,82653,-17547
C00627=-174479,-103807,-115834,-1877,80312,-17516
C00628=-174723,-101054,-114019,-1793,80601,-17598
C00629=-174059,-101482,-114177,-2021,80493,-17381
C00630=-175099,-100864,-114052,-1663,80716,-17725
C00631=-173219,-101718,-114202,-2308,80412,-17111
C00632=-174297,-103323,-108637,-11631,70926,-18463
C00633=-170332,-104420,-108349,-13314,70794,-17046
C00634=-174390,-105691,-110273,-11607,70709,-18474
C00635=-174377,-104937,-112785,-11492,72607,-18653
C00636=-190845,-100837,-124447,13698,93294,-33124
C00637=-206306,-116062,-120388,37359,88631,-50073
C00638=-215039,-120395,-106715,50971,83253,-62053
C00639=-215038,-119729,-104733,51036,82687,-62365
C00640=-214845,-117737,-104335,50959,83080,-62044
C00641=-214845,-116534,-100782,51086,82069,-62602
C00642=-215047,-118800,-102176,51129,81987,-62759
C00643=-215049,-119543,-104187,51057,82539,-62453
C00644=-215012,-122438,-115563,50746,86080,-60488
C00645=-160845,-113405,-113287,47121,77099,31472
C00646=-160851,-113463,-110064,47446,75709,30781
C00647=-161105,-114307,-109195,47677,75177,30385
C00648=-161122,-114371,-109216,47688,75170,30377
C00649=-115363,-119356,-110747,30444,52974,43110
C00650=-116247,-123536,-113883,31027,53106,42730
C00651=-160782,-112987,-114684,46949,77813,31850
C00652=-161690,-87231,-108001,36248,90547,80444
C00653=-156405,-91013,-102041,34922,83859,80351
C00654=-152529,-73393,-94338,33696,85968,82496
C00655=-158330,-83683,-104653,35339,89043,81248
C00656=-160758,-112853,-114863,36163,82877,78288
C00657=-160760,-113152,-111426,36317,81029,77674
C00658=-159491,-108015,-113138,31549,97627,78488
C00659=-160866,-112928,-114836,31527,96856,77736
C00660=-163914,-124233,-119408,29285,98886,76856
C00661=-164622,-129006,-121133,28240,99357,76613
C00662=-160757,-112482,-116558,30024,102576,77779
C00663=-160755,-111254,-119690,30396,104801,78387
C00664=-139139,-104942,-132434,5076,105021,81413
C00665=-120610,-140892,-128239,-26796,83300,73925
C00666=-124485,-139346,-124335,-26282,80622,73071
C00667=-128794,-174695,-130569,-28116,58521,76693
C00668=-123854,-173705,-127920,-33486,56775,79744
C00669=-127596,-155142,-123084,-28725,56836,77726
C00670=-128095,-155529,-122172,-29132,53686,78388
C00671=-128860,-155984,-126780,-25446,58633,74277
C00672=-138109,-135032,-133743,-8289,74304,51513
C00673=-203654,-125968,-124215,37381,73551,-30645
C00674=-201127,-103516,-110680,20461,62884,-59060
C00675=-201138,-104157,-107983,20829,61019,-59420
C00676=-208979,-113447,-103647,35969,52390,-64587
C00677=-207523,-116938,-104803,35675,50897,-64444
C00678=-203522,-124467,-107663,33692,47814,-63600
C00679=-203048,-125499,-107979,33578,47343,-63533
C00680=-201116,-104130,-107973,20816,61021,-59411
C00681=-201105,-103488,-110669,20449,62886,-59051
C00682=-198523,-119273,-121454,24683,77158,-64296
C00683=-174403,-100049,-121231,21877,99309,-62114
C00684=-174406,-102879,-118773,21681,96545,-62622
C00685=-198531,-152926,-120143,46630,71175,-78393
C00686=-201027,-150961,-118520,46868,72485,-79003
C00687=-203634,-147652,-117189,46113,74758,-79187
C00688=-204968,-146691,-116266,46227,75394,-79539
C00689=-174418,-104205,-117181,21599,94999,-62906
C00690=-174415,-101880,-119808,21752,97619,-62429
C00691=-185776,-93152,-118465,-1785,83350,-67432
C00692=-169060,-142396,-123848,-37084,49654,-60484
C00693=-174230,-113472,-108308,-34615,49911,-64397
C00694=-174247,-112967,-104740,-35556,48304,-63744
C00695=-204508,-109224,-105676,16537,47962,-87996
C00696=-204889,-112247,-105846,17210,46647,-88414
C00697=-205137,-117448,-106109,18144,44307,-89002
C00698=-205476,-118878,-106400,18590,43853,-89268
C00699=-202316,-128438,-104501,16790,32281,-90186
C00700=-174246,-112406,-102200,-36228,47262,-63291
C00701=-174229,-113129,-105847,-35265,48804,-63944
C00702=-182962,-136134,-123657,-29797,44727,-67038
C00703=-203654,-125968,-124215,37381,73551,-30645
C00704=-201127,-103516,-110680,20461,62884,-59060
C00705=-201138,-104157,-107983,20829,61019,-59420
C00706=-197142,-94471,-103147,18291,61982,-57680
C00707=-195983,-97109,-104177,17762,61047,-57388
C00708=-192692,-104164,-106885,16201,58502,-56495
C00709=-191828,-105876,-107504,15777,57855,-56246
C00710=-201116,-104130,-107973,20816,61021,-59411
C00711=-201105,-103488,-110669,20449,62886,-59051
C00712=-198523,-119273,-121454,24683,77158,-64296
C00713=-174403,-100049,-121231,21877,99309,-62114
C00714=-174406,-102879,-118773,21681,96545,-62622
C00715=-188779,-171638,-134697,28897,67939,-73565
C00716=-192229,-168597,-132843,29394,69543,-74545
C00717=-196575,-165255,-130680,29999,71416,-75803
C00718=-197254,-164985,-130459,30096,71662,-76012
C00719=-174418,-104205,-117181,21599,94999,-62906
C00720=-174415,-101880,-119808,21752,97619,-62429
C00721=-185776,-93152,-118465,-1785,83350,-67432
C00722=-169060,-142396,-123848,-37084,49654,-60484
C00723=-174230,-113472,-108308,-34615,49911,-64397
C00724=-174247,-112967,-104740,-35556,48304,-63744
C00725=-189487,-115301,-102458,-10134,35014,-67724
C00726=-189453,-118613,-102224,-10661,33197,-67437
C00727=-189517,-120543,-102067,-10903,32120,-67310
C00728=-189531,-122888,-102312,-11213,31079,-67147
C00729=-174246,-112406,-102200,-36228,47262,-63291
C00730=-175798,-117006,-109100,-34199,48210,-64559
C00731=-178617,-124532,-114828,-32467,46840,-65534
C00732=-210827,-121899,-127370,-35396,86436,-76908
C00733=-214505,-124636,-123608,-35577,86411,-76994
C00734=-214521,-124823,-120077,-35640,84542,-76397
C00735=-209595,-138372,-118962,-40572,76618,-76704
C00736=-215572,-134536,-117924,-37557,71164,-81051
C00737=-214545,-124844,-120083,-35636,84527,-76402
C00738=-214528,-124659,-123615,-35573,86395,-76999
C00739=-214596,-124890,-121786,-39550,96156,-78039
C00740=-214607,-124784,-118461,-39383,94595,-77461
C00741=-215336,-122839,-115954,-39308,93846,-77495
C00742=-215216,-123286,-113688,-39218,92622,-76995
C00743=-214785,-119888,-114308,-39371,94481,-77497
C00744=-214619,-124823,-118761,-39395,94718,-77513
C00745=-214540,-124430,-116246,-48349,86426,-68042
C00746=-214499,-123956,-126099,-48385,90728,-70182
C00747=-158797,-145907,-128305,-56145,74291,-56792
C00748=-118138,-117595,-113507,-59219,64127,-52420
C00749=-134091,-119062,-102284,-58108,50235,-52331
C00750=-134095,-117716,-98836,-59129,49460,-51612
C00751=-135589,-116107,-97216,-58736,48446,-51881
C00752=-133944,-119965,-109730,-11592,43893,-62364
C00753=-134860,-119489,-109370,-10824,43788,-62800
C00754=-134735,-119167,-109009,-10713,43511,-63435
C00755=-134110,-120442,-105586,-8081,38879,-71409
C00756=-134097,-120880,-107281,-7954,39689,-71484
C00757=-133538,-122024,-122159,-7272,48238,-71950
C00758=-134045,-120979,-109361,-39707,45136,-55893
C00759=-134048,-117179,-98466,-43015,41514,-53843
C00760=-133531,-117259,-97745,-41276,40690,-53975
C00761=-134198,-118862,-102182,-12962,37460,-61550
C00762=-134143,-118678,-102473,-12938,37734,-61565
C00763=-167359,-107040,-94607,43986,50437,-74743
C00764=-162364,-123197,-107171,35832,43944,-75497
C00765=-134045,-120979,-109361,-39707,45136,-55893
C00766=-132003,-121638,-109572,-41117,45917,-55073
C00767=-131002,-106489,-98392,-41164,47077,-55091
C00768=-131123,-103588,-88252,-50265,40796,-51296
C00769=-163242,-98975,-95762,18008,45953,-74760
C00770=-153405,-104865,-97946,10266,42608,-70493
C00771=-134148,-119761,-102793,-13034,37388,-61506
C00772=-126986,-126229,-93303,56145,28917,-85918
C00773=-131099,-132353,-104040,54087,33374,-85008
C00774=-133651,-114033,-99266,51853,45977,-77066
C00775=-134816,-132236,-131789,-6177,48808,-72548
C00776=-152519,-98596,-126841,-17039,86437,-59409
C00777=-167034,-82548,-116958,-26153,108191,-47353
C00778=-167227,-85698,-113927,-25595,104988,-46679
C00779=-155614,-79416,-105751,-37322,108167,-45505
C00780=-159401,-74916,-103736,-37095,107545,-46814
C00781=-167948,-62631,-97829,-36299,106456,-49792
C00782=-170767,-58288,-95591,-35952,106111,-50754
C00783=-180979,-58723,-101497,-23976,107062,-51805
C00784=-180909,-54943,-104050,-24554,110296,-52487
C00785=-168157,-75412,-102271,-33648,91006,-21456
C00786=-174012,-67106,-91297,-33471,82630,-14810
C00787=-175466,-61382,-85667,-32996,81659,-15067
C00788=-176048,-58561,-83401,-32769,81494,-15237
C00789=-213617,-47146,-82110,19258,88348,-36961
C00790=-192866,-61617,-91305,19873,90672,-32148
C00791=-185269,-67932,-94482,17568,87859,-30106
C00792=-154362,-96202,-104591,-19297,70625,-24481
C00793=-154503,-104813,-110762,-19306,69999,-24428
C00794=-155575,-73729,-96860,-32555,86012,-14938
C00795=-157088,-68154,-91284,-32096,84992,-15206
C00796=-157731,-66276,-89193,-31903,84490,-15302
C00797=-195536,-81793,-95810,17096,71410,-32670
C00798=-183377,-91714,-99996,11703,66886,-28896
C00799=-199796,-81518,-91231,35244,71315,-57262
C00800=-201423,-82172,-92479,35779,72324,-57601
C00801=-205660,-83542,-95477,37134,74990,-58446
C00802=-150225,-90058,-124320,-20069,81923,-14603
C00803=-88917,-116100,-126028,-29630,66347,39612
C00804=-48102,-114880,-112674,-35477,56596,75725
C00805=-53396,-105773,-101201,-33500,52497,74682
C00806=-53385,-105323,-98106,-34230,51099,75219
C00807=-48465,-101460,-95464,-40425,56724,79171
C00808=-72122,-108844,-98440,461,39847,55622
C00809=-53363,-105522,-99057,-19217,46878,60217
C00810=-53371,-105892,-101942,-18746,48378,59901
C00811=-53322,-113038,-104699,812,43724,42660
C00812=-53318,-112442,-102021,830,42382,42650
C00813=-53317,-112163,-100935,837,41857,42645
C00814=-53253,-112229,-97736,1547,37461,42516
C00815=-53300,-111445,-98358,1568,38246,42506
C00816=-51520,-115460,-104005,-179,39644,43460
C00817=-55761,-139961,-122674,-27476,66843,55729
C00818=-53542,-121644,-113892,-40363,83761,61539
C00819=-53523,-121175,-111327,-40444,82737,61941
C00820=-53533,-120846,-110023,-41635,87424,59647
C00821=-53533,-120798,-109834,-41636,87355,59676
C00822=-53529,-120315,-108043,-41648,86710,59935
C00823=-53536,-120580,-109029,-41640,87063,59791
C00824=-53556,-121151,-111460,-41628,87965,59422
C00825=-52633,-122748,-126719,-40391,89833,59612
C00826=-140119,-108661,-130674,-21165,82789,-25459
C00827=-161125,-123349,-120158,-18581,66270,-46079
C00828=-131164,-149034,-123827,-31550,65486,-33807
C00829=-140998,-169851,-126834,-7032,44376,-36345
C00830=-121609,-161923,-119940,-40371,51959,-24321
C00831=-116702,-163999,-110594,-61694,50034,-17487
C00832=-138878,-147559,-105015,-60087,46949,-25474
C00833=-144162,-146903,-104865,-58673,43866,-26892
C00834=-161212,-123488,-116538,-18871,64068,-45743
C00835=-161202,-123677,-120265,-18562,66156,-46089
C00836=-167124,-146469,-125858,32695,63076,-70922
C00837=-161220,-122264,-110536,44525,64077,-74742
C00838=-161219,-121375,-107584,44985,63095,-75224
C00839=-164956,-113819,-102428,48447,66739,-75134
C00840=-161214,-120895,-106203,44006,60818,-74436
C00841=-161480,-119432,-103853,44775,56123,-75022
C00842=-161477,-119788,-101535,47560,52624,-77093
C00843=-161197,-119682,-102993,46927,53134,-76618
C00844=-161197,-120736,-105876,46275,53998,-76117
C00845=-161177,-121556,-108554,35078,57327,-43050
C00846=-161177,-120932,-106617,35398,56609,-43319
C00847=-156320,-124656,-107064,29952,50956,-43105
C00848=-161176,-119594,-102910,36338,54666,-44181
C00849=-161179,-121157,-107284,34368,64565,-45309
C00850=-161179,-121533,-108462,34233,65010,-45160
C00851=-161180,-122193,-110741,33972,65899,-44866
C00852=-159909,-111206,-128347,-10927,59798,-43136
C00853=-174276,-119239,-128019,9099,73009,32604
C00854=-174287,-122281,-118814,9519,65873,32039
C00855=-174304,-122135,-115653,9666,64029,31878
C00856=-160412,-139818,-114717,-7630,47448,36959
C00857=-152446,-94935,-106365,-29486,98792,40063
C00858=-160237,-131582,-118994,-28233,86388,40212
C00859=-174317,-121775,-113110,-33515,107538,43031
C00860=-174312,-121937,-114098,-33622,107981,42892
C00861=-174299,-122214,-116525,-33911,109120,42531
C00862=-174287,-119835,-127268,-36019,115609,40290
C00863=-174287,-120021,-127206,9145,72119,32532
C00864=-174287,-120021,-127206,9145,72119,32532
C00865=-173736,-117333,-114872,9262,65925,32245
C00866=-174960,-111711,-111152,9771,66659,31859
C00867=-176831,-126585,-121826,-8311,79476,36809
C00868=-157010,-133467,-117360,-32643,99223,56368
C00869=-157552,-135759,-118018,-32604,98358,56401
C00870=-154345,-130153,-124672,-33336,105500,55567
C00871=-134844,-151987,-134250,-26337,102553,60683
C00872=-146682,-141770,-131473,-27794,101884,56245
C00873=-146682,-141770,-131473,15257,98468,53705
C00874=-102938,-141770,-131473,49664,98468,53705
C00875=-102938,-145417,-131473,49512,65454,53705
C00876=-103656,-129714,-109721,51674,62395,51470
C00877=-103209,-138986,-102320,63457,51189,43454
C00878=-119944,-123339,-96652,64718,84974,57690
C00879=-120711,-153122,-104212,65541,80717,53119
C00880=-119902,-122365,-94692,64738,95453,62634
C00881=-116435,-131456,-112749,56730,96510,65994
C00882=-116383,-133294,-113279,56655,96128,65766
C00883=-84454,-125099,-129012,35107,90636,33075
C00884=-15972,-110889,-128286,-10965,59905,-43045
C00885=-12667,-135547,-130714,31270,45596,0
C00886=-9315,-159766,-119262,-3212,6219,55552
C00887=-157761,-135547,-130714,31270,45596,-69143
C00888=-154472,-113934,-104337,41712,51336,-70449
C00889=-149832,-108771,-100172,39130,49259,-68869
C00890=-148058,-106656,-98467,38074,48499,-68236
C00891=-148062,-106275,-96666,38578,47777,-68578
C00892=-148058,-106656,-98467,38074,48499,-68236
C00893=-147997,-106381,-96958,38469,47847,-68508
C00894=-145894,-104035,-96109,36815,47477,-67498
C00895=-147997,-106381,-96958,38469,47847,-68508
C00896=-154410,-113635,-102825,42095,50721,-70729
C00897=-154342,-120637,-107041,25827,48602,-38771
C00898=-150292,-111683,-102360,22573,48994,-36710
C00899=-148798,-108210,-100464,21373,49171,-35962
C00900=-146664,-105787,-99597,19708,49308,-34937
C00901=-146949,-106220,-99797,19932,49282,-35074
C00902=-147721,-103636,-97533,20478,49410,-35405
C00903=-146949,-106220,-99797,19932,49282,-35074
C00904=-152261,-118724,-106469,24248,48548,-37770
C00905=-148295,-114597,-117137,-6490,60568,-69086
C00906=-147868,-109631,-111600,-6790,59752,-68875
C00907=-147704,-107727,-109395,-6911,59390,-68790
C00908=-147708,-107860,-107783,-6984,58336,-68724
C00909=-147704,-107727,-109395,-6911,59390,-68790
C00910=-147723,-107760,-107968,-6963,58499,-68740
C00911=-147306,-102596,-106094,-7098,60024,-68678
C00912=-147723,-107760,-107968,-6963,58499,-68740
C00913=-148315,-114751,-115749,-6537,59639,-69038
C00914=-148355,-114889,-117236,-6461,60467,-69101
C00915=-147925,-109892,-111692,-6763,59663,-68890
C00916=-147761,-107977,-109485,-6884,59305,-68805
C00917=-147764,-108104,-107870,-6957,58254,-68739
C00918=-147777,-108153,-108078,-6942,58354,-68751
C00919=-147358,-102980,-106206,-7078,59886,-68688
C00920=-147777,-108153,-108078,-6942,58354,-68751
C00921=-148373,-115211,-115873,-6515,59468,-69049
C00922=-147696,-122269,-111871,-35505,39043,-51945
C00923=-147690,-118447,-100224,-39719,34874,-49579
C00924=-148491,-109409,-94254,-38171,35277,-50420
C00925=-148787,-105724,-91002,-38010,35060,-50504
C00926=-148789,-105382,-89977,-38411,34697,-50285
C00927=-149058,-101689,-89016,-37046,35623,-51030
C00928=-149145,-100783,-88679,-36755,35795,-51189
C00929=-149058,-101689,-89016,-37046,35623,-51030
C00930=-145777,-99657,-88811,-39022,37803,-49998
C00931=-148139,-100407,-89095,-37251,36591,-50936
C00932=-145777,-99657,-88811,-39022,37803,-49998
C00933=-147690,-118447,-100224,-39719,34874,-49579
C00934=-128033,-128545,-103748,-39689,32513,-43973
C00935=-128383,-118409,-97778,-37905,33566,-44930
C00936=-128511,-114277,-94563,-37658,33626,-45064
C00937=-128512,-113804,-93446,-38069,33271,-44843
C00938=-129119,-111006,-93029,-36452,33958,-45715
C00939=-129434,-109852,-92636,-35862,34111,-46033
C00940=-128358,-113721,-93936,-37885,33613,-44941
C00941=-176216,-70111,-78093,55162,70856,-80763
C00942=-174311,-70781,-78417,54616,69674,-80426
C00943=-176216,-70111,-78093,55162,70856,-80763
C00944=-181747,-69996,-81392,56304,75271,-81045
C00945=-178033,-77165,-93769,42680,75059,-77098
C00946=-164745,-109340,-116699,-3009,62053,-68278
C00947=-145851,-112599,-102075,-47717,41998,-56322
C00948=-148044,-104803,-96379,-45883,41204,-57334
C00949=-148864,-101708,-93474,-45490,40644,-57533
C00950=-148866,-101457,-92299,-45986,40221,-57239
C00951=-148863,-101834,-94104,-45225,40876,-57690
C00952=-145127,-99228,-91361,-47944,42572,-56214
C00953=-147466,-100038,-91670,-46636,41186,-56907
C00954=-145127,-99228,-91361,-47944,42572,-56214
C00955=-146129,-107372,-95667,-48598,40993,-55782
C00956=-148216,-109089,-93488,-49289,38371,-55335
C00957=-148344,-107837,-93052,-48851,38553,-55585
C00958=-147906,-112054,-94498,-50363,37947,-54724
C00959=-145851,-112599,-102075,-47717,41998,-56322
C00960=-158250,-140903,-124067,-47621,67451,-49320
C00961=-161740,-133075,-117656,-46661,65672,-50232
C00962=-162335,-130592,-114553,-46699,64919,-50156
C00963=-162276,-129951,-113381,-46845,64676,-49998
C00964=-160420,-132544,-115533,-47350,65644,-49520
C00965=-135901,-74424,-73697,-74364,100921,-31256
C00966=-137788,-75503,-74147,-74218,99532,-31324
C00967=-138769,-76027,-74362,-74146,98812,-31363
C00968=-135901,-74424,-73697,-74364,100921,-31256
C00969=-149282,-147643,-98518,-79858,51263,-26133
C00970=-149394,-146891,-98381,-79629,51249,-26315
C00971=-148448,-152811,-99407,-81432,51428,-24854
C00972=-139735,-166147,-105854,-82069,56849,-22658
C00973=-180438,-97574,-115199,-33764,102267,52414
C00974=-189965,-108899,-115705,-31971,94091,51156
C00975=-190633,-110068,-115194,-31831,93066,51189
C00976=-190637,-110288,-114404,-31804,92551,51332
C00977=-190629,-109833,-115910,-31859,93547,51055
C00978=-186867,-102382,-113240,-32521,96788,51574
C00979=-187005,-102964,-110979,-32373,95300,51952
C00980=-188888,-106610,-112304,-32065,93703,51681
C00981=-187005,-102964,-110979,-32373,95300,51952
C00982=-188021,-107681,-112675,-32159,93748,52003
C00983=-189590,-103281,-111094,-32025,94271,51250
C00984=-188021,-107681,-112675,-32159,93748,52003
C00985=-180438,-97574,-115199,-33764,102267,52414
C00986=-185735,-83978,-109774,-33564,103394,50026
C00987=-199988,-77820,-108712,11582,98175,-38155
C00988=-204749,-56978,-92496,29836,109182,-47433
C00989=-202460,-56662,-91339,29422,107990,-46925
C00990=-201413,-57385,-91726,29256,107546,-46663
C00991=-201611,-57041,-91542,29296,107663,-46703
C00992=-201611,-58240,-90431,29070,106521,-47008
C00993=-203359,-50274,-87822,29763,109247,-46906
C00994=-195470,-25798,-72981,29209,109868,-43903
C00995=-195013,-27562,-73704,29036,109327,-43888
C00996=-194283,-28250,-74172,28893,109053,-43704
C00997=-194480,-28066,-74047,28932,109127,-43754
C00998=-194480,-29296,-73135,28708,108075,-44034
C00999=-195605,-24849,-71507,29147,109538,-44038
C01000=-191110,-5546,-57842,28597,109561,-42465
C01001=-192519,-3768,-54500,33008,111368,-41387
C01002=-191992,-5303,-55742,32912,111174,-41254
C01003=-192059,-5108,-55586,32924,111198,-41271
C01004=-192059,-6294,-54683,32651,110210,-41583
C01005=-192882,-2296,-53893,33162,111810,-41382
C01006=-203365,-15491,-64400,34648,115083,-44256
C01007=-218411,-26661,-75493,58573,107247,-46176
C01008=-145332,-87800,-123084,4045,108310,15756
C01009=-109199,-104290,-129101,-21867,105305,43874
C01010=-112610,-115777,-129409,-14908,94573,36374
C01011=-117115,-112620,-124614,-14006,92529,35127
C01012=-118008,-112320,-123068,-13816,91609,34934
C01013=-118007,-112900,-122267,-13806,90840,35020
C01014=-118044,-112536,-122505,-13803,91159,34973
C01015=-118576,-105776,-120168,-13731,93052,34586
C01016=-118044,-112536,-122505,-13803,91159,34973
C01017=-125955,-111499,-122045,-12179,90192,32457
C01018=-127333,-111877,-122174,-11884,89885,32033
C01019=-124755,-111115,-121914,-12435,90480,32824
C01020=-119624,-116552,-128230,-13509,92325,34321
C01021=-117231,-121833,-124467,-22052,85463,28755
C01022=-122341,-114124,-118662,-20866,84531,27121
C01023=-123318,-113111,-117155,-20643,83910,26885
C01024=-123641,-113323,-116249,-20585,83205,26892
C01025=-123595,-112804,-116375,-20585,83540,26851
C01026=-123397,-106736,-114247,-20589,85286,26623
C01027=-123595,-112804,-116375,-20585,83540,26851
C01028=-116023,-114044,-115764,-22346,84523,29358
C01029=-117346,-116777,-115957,-22098,82979,29171
C01030=-118867,-116723,-116143,-21757,82713,28674
C01031=-116293,-116772,-115815,-22329,83179,29512
C01032=-117231,-121833,-124467,-22052,85463,28755
C01033=-154726,-134692,-133300,19029,79240,32627
C01034=-155157,-123239,-125350,19102,80279,32639
C01035=-155214,-122106,-123677,19140,79867,32554
C01036=-155216,-122330,-122794,19175,79245,32454
C01037=-155272,-122641,-123186,19186,79334,32449
C01038=-154565,-115790,-120970,18882,81218,32994
C01039=-155272,-122449,-123985,19155,79894,32538
C01040=-110972,-119209,-121408,-15853,79302,48266
C01041=-109086,-133769,-122042,-16854,72857,49812
C01042=-111848,-135958,-122676,-16103,71595,48979
C01043=-109086,-133769,-122042,-16854,72857,49812
C01044=-108592,-130707,-130810,-16554,79646,49045
C01045=-120610,-122471,-119242,-21572,81234,22537
C01046=-120610,-122484,-118172,-21604,80613,22649
C01047=-120610,-122391,-116483,-21658,79689,22817
C01048=-120610,-122419,-116833,-21647,79876,22783
C01049=-120610,-122423,-116832,-21647,79874,22783
C01050=-120610,-122419,-116833,-21647,79876,22783
C01051=-120610,-122416,-116761,-21649,79836,22790
C01052=-120610,-122436,-116768,-21650,79830,22791
C01053=-120610,-122416,-116761,-21649,79836,22790
C01054=-120611,-122370,-120508,-21535,82009,22397
C01055=-120500,-119354,-126515,-17332,87675,17755
C01056=-155157,-123239,-125350,19102,80279,32639
C01057=-155214,-122106,-123677,19140,79867,32554
C01058=-155216,-122330,-122794,19175,79245,32454
C01059=-155272,-122641,-123186,19186,79334,32449
C01060=-154565,-115790,-120970,18882,81218,32994
C01061=-155272,-122449,-123985,19155,79894,32538
C01062=-110972,-119209,-121408,-15853,79302,48266
C01063=-109086,-133769,-122042,-16854,72857,49812
C01064=-111848,-135958,-122676,-16103,71595,48979
C01065=-109086,-133769,-122042,-16854,72857,49812
C01066=-108592,-130707,-130810,-16554,79646,49045
C01067=-120611,-118687,-129075,-3134,90000,4412
C01068=-120611,-121772,-123926,-3138,85252,4531
C01069=-120611,-122092,-122744,-3141,84362,4553
C01070=-120611,-122362,-121169,-3146,83256,4581
C01071=-120611,-122286,-121724,-3144,83636,4571
C01072=-120611,-122290,-121724,-3144,83633,4571
C01073=-120611,-122286,-121724,-3144,83636,4571
C01074=-120611,-121006,-125813,-3134,86805,4492
C01075=-120621,-113915,-131911,-13153,116790,34478
C01076=-136832,-143297,-133894,-19017,104291,40845
C01077=-187686,-122249,-118318,-34521,102174,42234
C01078=-187703,-122088,-115580,-34298,100833,42653
C01079=-187707,-122010,-114917,-34250,100525,42749
C01080=-187713,-121734,-113169,-34135,99743,42991
C01081=-187707,-122010,-114917,-34250,100525,42749
C01082=-187770,-121697,-112491,-32279,113674,44764
C01083=-187767,-121692,-112491,-32279,113678,44765
C01084=-187770,-121697,-112491,-32279,113674,44764
C01085=-187667,-121438,-112064,-34928,84963,41689
C01086=-187673,-121448,-112068,-34927,84958,41688
C01087=-187667,-121438,-112064,-34928,84963,41689
C01088=-187641,-121360,-124129,-34919,91154,39753
C01089=-178673,-119471,-127738,-23493,103847,53429
C01090=-160878,-120510,-126471,-37,121976,81968
C01091=-160881,-121699,-123664,-37,119637,81967
C01092=-160883,-121991,-122485,-37,118762,81967
C01093=-160886,-122244,-120905,-37,117660,81966
C01094=-160884,-122111,-121864,-37,118318,81967
C01095=-160882,-122100,-121862,-36,118322,81968
C01096=-160884,-122111,-121864,-37,118318,81967
C01097=-160879,-120821,-125908,-37,121469,81968
C01098=-160879,-120821,-131564,-37,121469,81968
C01099=-157394,-128671,-131753,738,117538,83283
C01100=-158801,-138021,-132727,409,113343,82737
C01101=-158801,-138035,-132347,409,113101,82737
C01102=-158801,-138034,-131509,408,112586,82736
C01103=-158801,-138039,-131833,408,112783,82736
C01104=-160693,-149427,-134985,6,108877,82039
C01105=-160612,-153549,-136083,24,107435,82069
C01106=-159125,-144348,-133603,336,110634,82611
C01107=-199963,-104116,-119881,11013,127404,83152
C01108=-204692,-116225,-118816,8637,121169,80600
C01109=-203581,-121519,-120530,8810,119404,80895
C01110=-204849,-113790,-122122,8953,124435,80816
C01111=-166129,-114439,-129167,13521,133132,-54375
C01112=-82387,-124374,-130385,21792,102809,-55833
C01113=-37550,-124758,-124791,27166,84975,-54517
C01114=-35933,-124831,-122904,26864,83389,-54284
C01115=-35589,-124875,-121597,26827,82538,-54351
C01116=-35584,-124889,-121174,26839,82296,-54405
C01117=-35764,-126387,-121953,26892,82093,-54519
C01118=-31633,-125451,-121673,25972,81076,-53208
C01119=-35764,-126387,-121953,26892,82093,-54519
C01120=-46981,-157328,-126723,35790,81436,-33730
C01121=-42905,-153934,-122174,35701,78867,-32870
C01122=-42758,-143813,-119569,35389,81762,-31868
C01123=-42905,-153934,-122174,35701,78867,-32870
C01124=-53188,-117519,-120731,36414,97747,-30962
C01125=-95179,-109851,-129540,3422,106316,17944
C01126=-143691,-100776,-119079,-26047,122130,73021
C01127=-146029,-112499,-120098,-24937,116556,73463
C01128=-147204,-116618,-119576,-24569,113992,73590
C01129=-147487,-116577,-118677,-24502,113425,73607
C01130=-146967,-116625,-120319,-24630,114475,73574
C01131=-147345,-121113,-121824,-24401,113105,73737
C01132=-146899,-128254,-123879,-23878,111030,74376
C01133=-147345,-121113,-121824,-24401,113105,73737
C01134=-118081,-135478,-120686,-30293,109901,65237
C01135=-118366,-136707,-118609,-29972,108136,65614
C01136=-120887,-140213,-119894,-30302,106351,65070
C01137=-118366,-136707,-118609,-29972,108136,65614
C01138=-117820,-130449,-123242,-31209,113594,64262
C01139=-93926,-103398,-125362,-18301,106221,39936
C01140=-72688,-110808,-124077,-7134,85250,24096
C01141=-75848,-101444,-116923,-6191,85411,23073
C01142=-76170,-100985,-115528,-6097,84767,23002
C01143=-76167,-101481,-114835,-6104,84090,23035
C01144=-78739,-96930,-113773,-5320,85595,22140
C01145=-79843,-95445,-113201,-4985,85938,21775
C01146=-77748,-98228,-114268,-5620,85298,22470
C01147=-140085,-104632,-109249,40944,98797,-6712
C01148=-140263,-103640,-106572,40817,98007,-7102
C01149=-137942,-102173,-106029,40697,97269,-6378
C01150=-140263,-103640,-106572,40817,98007,-7102
C01151=-135988,-101428,-112112,41019,99549,-4631
C01152=-141957,-83285,-117139,12315,91699,6710
C01153=-161957,-129781,-122866,-20018,67926,12328
C01154=-166016,-109699,-113650,-17211,72980,10098
C01155=-166795,-105246,-111748,-16434,74862,9605
C01156=-165677,-113012,-111900,-18316,68836,10778
C01157=-162725,-116093,-113629,-19548,69016,11850
C01158=-162651,-107484,-110669,-19284,71494,11460
C01159=-162725,-116093,-113629,-19548,69016,11850
C01160=-155151,-112727,-112486,-22270,71877,14160
C01161=-155120,-113819,-110277,-22518,70103,14518
C01162=-159000,-114269,-110433,-21107,68960,13264
C01163=-155120,-113819,-110277,-22518,70103,14518
C01164=-155137,-138999,-124748,-23105,66364,15269
C01165=-81055,-115973,-127517,23586,109336,-64560
C01166=-76492,-127739,-126040,22738,101683,-64421
C01167=-76072,-128597,-125529,22671,100870,-64425
C01168=-76065,-128640,-125326,22657,100732,-64448
C01169=-76072,-128576,-125785,22685,101025,-64394
C01170=-82641,-146978,-130130,22016,96499,-67668
C01171=-81130,-155003,-132256,21951,93476,-67670
C01172=-82641,-146978,-130130,22016,96499,-67668
C01173=-84000,-144678,-127518,21929,96467,-68175
C01174=-84000,-143983,-126065,21900,95967,-68269
C01175=-83327,-146231,-127404,21916,95478,-68108
C01176=-88356,-135439,-132684,22407,104994,-68175
C01177=-104080,-128245,-132212,-31995,84146,-22143
C01178=-106783,-105266,-117364,-31197,85468,-23533
C01179=-107129,-103609,-115494,-31111,85090,-23558
C01180=-107127,-104217,-114421,-31144,84251,-23329
C01181=-107044,-104571,-114816,-31164,84333,-23320
C01182=-107880,-99055,-112779,-30885,85404,-23924
C01183=-107044,-104571,-114816,-31164,84333,-23320
C01184=-105114,-115284,-123193,-31689,84721,-22698
C01185=-105208,-113465,-123990,-31624,85910,-23065
C01186=-106823,-104635,-117017,-31184,85549,-23570
C01187=-107122,-103295,-115264,-31113,85109,-23561
C01188=-107121,-103855,-114286,-31142,84342,-23351
C01189=-107087,-104437,-114776,-31151,84356,-23343
C01190=-107921,-98925,-112738,-30873,85426,-23945
C01191=-107087,-104437,-114776,-31151,84356,-23343
C01192=-105701,-116384,-125830,-31502,85418,-23114
C01193=-79137,-116524,-127291,-7118,77084,38210
C01194=-66518,-158449,-133200,-8588,59166,50817
C01195=-70166,-147728,-127011,-6864,60501,49298
C01196=-71549,-143558,-123868,-6244,60595,48757
C01197=-71544,-142942,-122687,-6271,60188,48782
C01198=-71412,-140542,-122600,-6259,61371,48766
C01199=-74130,-137647,-121783,-5023,62161,47690
C01200=-71412,-140542,-122600,-6259,61371,48766
C01201=-59221,-85077,-106862,-19044,97138,55247
C01202=-59772,-90133,-108950,-18878,95774,55276
C01203=-59221,-85077,-106862,-19044,97138,55247
C01204=-65406,-128676,-128270,-8670,80773,42177
C01205=-57064,-112054,-129147,-2862,108793,29097
C01206=-70948,-123089,-127271,10962,111372,-380
C01207=-67644,-116564,-123033,11394,111660,848
C01208=-67644,-116773,-122597,11361,111292,811
C01209=-67644,-116291,-123546,11437,112109,893
C01210=-70770,-123262,-125779,10903,110357,-412
C01211=-70770,-123588,-124717,10837,109552,-488
C01212=-69306,-120453,-123728,11077,110342,115
C01213=-70770,-123283,-125719,10898,110311,-416
C01214=-70770,-119886,-130778,11344,115083,53
C01215=-68413,-122856,-123349,22437,117236,58
C01216=-67404,-122631,-120786,22344,115611,123
C01217=-67401,-122683,-120099,22253,115193,37
C01218=-67283,-122594,-120333,22317,115338,115
C01219=-65261,-118175,-118917,23034,116088,1096
C01220=-67283,-122594,-120333,22317,115338,115
C01221=-70820,-123560,-126018,22187,119059,-540
C01222=-59587,-128850,-129971,-18356,103459,48793
C01223=-60648,-112549,-116046,-37363,97913,74718
C01224=-66648,-121539,-115269,-36526,91263,74498
C01225=-69624,-125916,-115212,-36242,88151,74300
C01226=-69624,-125773,-114639,-36242,87924,74374
C01227=-69624,-125814,-114800,-36242,87987,74354
C01228=-70738,-127677,-115368,-36152,87024,74211
C01229=-69624,-125814,-114800,-36242,87987,74354
C01230=-61556,-115340,-115782,-37136,96245,74919
C01231=-93863,-107857,-129738,-18786,98098,27923
C01232=-113340,-105978,-120535,-17383,92037,15860
C01233=-116256,-99504,-115214,-16745,91512,14962
C01234=-117355,-97038,-113094,-16498,91266,14630
C01235=-124053,-106600,-116618,-14934,87391,12894
C01236=-123019,-109757,-118902,-15179,87365,13243
C01237=-120254,-118381,-124729,-15823,87055,14212
C01238=-121076,-118719,-112405,-41381,81563,9211
C01239=-125328,-110839,-107644,-40465,80446,7775
C01240=-126920,-107772,-105722,-40091,80023,7243
C01241=-122279,-105715,-102241,-45382,81605,7865
C01242=-118123,-103314,-98388,-50429,83325,8212
C01243=-115452,-99808,-95169,-50805,84680,8860
C01244=-113598,-101964,-96694,-51043,85596,9323
C01245=-108732,-107177,-100380,-51565,88044,10518
C01246=-131658,-113091,-133069,-11905,90618,-13395
C01247=-155934,-143784,-122811,23124,58745,-32427
C01248=-151507,-132468,-117411,20635,59886,-30339
C01249=-149876,-128251,-115276,19729,60288,-29596
C01250=-151213,-128323,-114307,20456,60014,-30191
C01251=-146890,-120795,-114089,13688,65901,-25886
C01252=-142734,-111238,-112703,7950,73001,-22079
C01253=-143750,-114926,-115045,8343,72653,-22456
C01254=-146492,-125018,-121022,9420,71459,-23506
C01255=-146459,-122334,-129315,9145,77857,-23007
C01256=-118526,-115013,-133262,8809,105739,-46794
C01257=-93674,-118800,-129721,8134,120991,-68616
C01258=-93669,-120967,-127104,7892,118292,-68817
C01259=-94465,-127736,-127937,7493,115415,-69310
C01260=-101667,-152205,-134731,5550,107657,-72408
C01261=-93660,-121042,-127131,7893,118270,-68815
C01262=-93665,-118880,-129750,8134,120967,-68614
C01263=-98446,-113408,-116165,41475,93741,-73013
C01264=-95217,-118830,-115137,40946,89638,-73223
C01265=-92806,-121560,-115150,40665,87459,-73017
C01266=-95954,-130241,-115077,41081,85472,-75169
C01267=-96936,-125131,-114749,41104,87782,-74702
C01268=-101504,-121000,-116278,41571,92256,-74948
C01269=-100864,-122088,-112493,43204,76282,-71688
C01270=-96953,-122826,-110054,42689,72984,-71279
C01271=-94247,-124338,-109802,42269,70974,-70864
C01272=-94193,-123974,-108080,42453,70297,-71131
C01273=-95642,-121622,-108630,42447,72155,-71017
C01274=-100864,-121830,-111367,43291,75868,-71867
C01275=-131033,-115476,-133015,2815,101744,-74384
C01276=-151471,-119125,-123137,-34971,103386,-73225
C01277=-162012,-101235,-114016,-37763,108592,-75954
C01278=-165297,-105997,-114400,-37202,105452,-76208
C01279=-161279,-107047,-112450,-36906,105725,-74600
C01280=-157962,-101866,-111865,-37402,108959,-74341
C01281=-155898,-93647,-112180,-38609,113341,-75115
C01282=-93674,-112333,-133466,8753,126560,-68151
C01283=-93674,-118800,-129721,8134,120991,-68616
C01284=-93669,-120967,-127104,7892,118292,-68817
C01285=-93667,-121558,-126026,7814,117333,-68886
C01286=-93663,-121536,-126144,7822,117416,-68879
C01287=-93639,-121762,-126135,7818,117296,-68878
C01288=-93680,-121434,-126040,7817,117406,-68885
C01289=-93660,-121042,-127131,7893,118270,-68815
C01290=-93665,-118880,-129750,8134,120967,-68614
C01291=-98446,-113408,-116165,41475,93741,-73013
C01292=-93996,-117843,-114815,40802,89312,-72817
C01293=-91343,-117266,-113836,40455,87860,-72224
C01294=-92137,-119395,-114109,40564,87510,-72703
C01295=-95072,-126184,-113786,40951,86041,-74561
C01296=-95071,-125918,-112907,40977,85731,-74679
C01297=-96936,-125131,-114749,41104,87782,-74702
C01298=-101504,-121000,-116278,41571,92256,-74948
C01299=-100864,-122088,-112493,43204,76282,-71688
C01300=-95643,-121963,-109784,42340,72556,-70846
C01301=-93677,-120964,-108398,41948,71358,-70433
C01302=-93599,-120925,-107098,42100,70733,-70661
C01303=-95642,-121622,-108630,42447,72155,-71017
C01304=-100864,-121830,-111367,43291,75868,-71867
C01305=-131033,-115476,-133015,2815,101744,-74384
C01306=-151471,-119125,-123137,-34971,103386,-73225
C01307=-162012,-101235,-114016,-37763,108592,-75954
C01308=-163593,-104354,-113811,-37340,106547,-75879
C01309=-162938,-104376,-113793,-37349,106803,-75692
C01310=-158829,-104862,-111593,-37019,107224,-74083
C01311=-157962,-101866,-111865,-37402,108959,-74341
C01312=-155898,-93647,-112180,-38609,113341,-75115
C01313=-179206,-139250,-107986,-62075,77828,-66561
C01314=-185232,-138953,-105140,-62379,73225,-66913
C01315=-187696,-139015,-104542,-62453,71468,-67163
C01316=-187702,-137665,-102648,-62587,71237,-66963
C01317=-185238,-138055,-103864,-62461,73065,-66778
C01318=-179211,-138396,-106727,-62132,77661,-66424
C01319=-179188,-148562,-121526,-61524,79591,-68010
C01320=-184417,-115822,-131978,-19629,107310,7500
C01321=-190427,-134899,-136820,8574,116374,78562
C01322=-188066,-120573,-128029,9218,118052,79593
C01323=-191610,-147357,-136376,6897,103791,75181
C01324=-187795,-119828,-126345,9210,117376,79639
C01325=-187841,-121664,-124728,-2971,114560,78170
C01326=-187942,-121398,-126015,-3016,115485,78109
C01327=-187937,-119495,-128851,-3098,118205,78035
C01328=-176042,-128909,-129640,-7380,110692,58022
C01329=-187833,-113452,-115854,-34994,105139,41767
C01330=-187847,-113781,-113588,-34722,103839,42187
C01331=-187853,-113844,-112659,-34623,103335,42348
C01332=-187856,-113866,-111596,-34519,102780,42525
C01333=-187851,-113844,-112538,-34611,103274,42368
C01334=-187836,-113627,-114840,-34866,104547,41960
C01335=-186756,-108501,-120882,-36201,110201,40487
C01336=-150585,-129060,-123753,-46684,114085,-39870
C01337=-134046,-137019,-115206,-49635,112096,-74674
C01338=-134033,-140586,-110307,-48065,108843,-72866
C01339=-134037,-138671,-107458,-47843,108316,-72589
C01340=-133950,-137111,-106105,-47812,108341,-72556
C01341=-133930,-150358,-126108,1173,113974,-57522
C01342=-134040,-150029,-126001,1133,114079,-57562
C01343=-134505,-148512,-125722,2741,114238,-57140
C01344=-137673,-151162,-132623,1623,117206,-58299
C01345=-106012,-107394,-121753,14018,130776,-44816
C01346=-106669,-102485,-112824,13121,127987,-45519
C01347=-97512,-96218,-110425,14566,129183,-82759
C01348=-98864,-105619,-112306,13303,125832,-83842
C01349=-106150,-109468,-113796,12766,125107,-45727
C01350=-105474,-116823,-114648,29161,97726,-33837
C01351=-134074,-146851,-118858,40485,90771,-46834
C01352=-141855,-151854,-132376,33568,89282,-32323
C01353=-173958,-148748,-133240,11874,65312,15203
C01354=-187653,-128002,-123664,-7056,57779,46476
C01355=-188071,-112180,-99768,1790,31671,46486
C01356=-188092,-111455,-97340,1875,30550,46442
C01357=-187851,-111485,-96835,1581,30220,46589
C01358=-187792,-110201,-93997,1555,29133,46605
C01359=-187737,-110060,-93474,1490,28882,46636
C01360=-187785,-109075,-90961,1604,27844,46576
C01361=-188106,-109627,-92159,2030,28303,46362
C01362=-188086,-110531,-94662,1935,29378,46411
C01363=-188086,-114129,-114927,1479,39995,46659
C01364=-201470,-41376,-102585,19941,97743,-57993
C01365=-197439,-2624,-49840,39121,107911,-51008
C01366=-168348,92819,48556,27514,116832,-48709
C01367=-170146,82769,36005,28011,119675,-48673
C01368=-172466,59662,8523,30747,114377,-38085
C01369=-173361,44293,-8668,31536,116980,-37634
C01370=-173326,42548,-10417,31798,119739,-39927
C01371=-173293,31446,-22173,31559,124382,-42741
C01372=-170045,43132,-9775,28753,130915,-51393
C01373=-186843,33187,-28183,45340,118495,-56566
C01374=-187270,22965,-40018,42118,113549,-44205
C01375=-164927,12374,-50848,37497,97302,26684
C01376=-160848,-52651,-98971,6904,73590,44156
C01377=-187933,-111679,-98706,-278,30585,46526
C01378=-187953,-110958,-96368,-260,29517,46517
C01379=-188171,-110591,-95666,34,29272,46369
C01380=-188111,-109885,-93130,-50,28074,46412
C01381=-188090,-109778,-92606,-82,27808,46427
C01382=-188055,-108797,-90194,-133,26826,46455
C01383=-187968,-109087,-91174,-258,27282,46516
C01384=-187948,-109974,-93584,-278,28309,46526
C01385=-190713,-138118,-122139,3147,45685,54861
C01386=-188097,-104568,-127563,3199,90457,72619
C01387=-188112,-108983,-124849,3203,86524,72515
C01388=-196049,-130715,-128058,11352,73875,69900
C01389=-193131,-119078,-125609,7963,80164,71095
C01390=-187364,-124777,-127140,2732,76642,72458
C01391=-191510,-130298,-128202,6704,73471,71168
C01392=-188153,-109076,-124888,3215,86502,72501
C01393=-188138,-104664,-127604,3212,90434,72606
C01394=-187898,-111965,-120493,-16766,69565,69566
C01395=-187918,-113285,-117348,-17044,67055,69927
C01396=-188336,-115132,-116370,-17036,65483,70009
C01397=-188181,-112945,-115606,-17029,66143,69965
C01398=-188166,-113080,-115592,-17048,66072,69982
C01399=-187991,-112297,-115306,-17102,66325,70009
C01400=-187944,-113344,-117352,-17035,67023,69922
C01401=-187924,-112030,-120500,-16757,69531,69561
C01402=-180038,-109975,-126789,-2440,82512,-7441
C01403=-174468,-102021,-118148,-1871,82653,-17547
C01404=-174479,-103807,-115834,-1877,80312,-17516
C01405=-175021,-104384,-114967,-1695,79470,-17680
C01406=-174783,-104250,-115053,-1777,79597,-17606
C01407=-174170,-106690,-109656,-11758,69864,-18312
C01408=-172833,-107431,-109671,-12341,69693,-17819
C01409=-174390,-105691,-110273,-11607,70709,-18474
C01410=-174377,-104937,-112785,-11492,72607,-18653
C01411=-190845,-100837,-124447,13698,93294,-33124
C01412=-206306,-116062,-120388,37359,88631,-50073
C01413=-215039,-120395,-106715,50971,83253,-62053
C01414=-215038,-119729,-104733,51036,82687,-62365
C01415=-215037,-119445,-103934,51064,82464,-62488
C01416=-215047,-118488,-101366,51160,81769,-62880
C01417=-215047,-118800,-102176,51129,81987,-62759
C01418=-215049,-119543,-104187,51057,82539,-62453
C01419=-215012,-122438,-115563,50746,86080,-60488
C01420=-160845,-113405,-113287,47121,77099,31472
C01421=-160851,-113463,-110064,47446,75709,30781
C01422=-161282,-114943,-109409,47754,75135,30277
C01423=-161254,-114846,-109376,47745,75139,30294
C01424=-160788,-113231,-109982,47419,75724,30819
C01425=-160782,-112987,-114684,46949,77813,31850
C01426=-161690,-87231,-108001,36248,90547,80444
C01427=-156210,-91223,-102127,34873,83736,80390
C01428=-152348,-73560,-94415,33644,85868,82536
C01429=-158330,-83683,-104653,35339,89043,81248
C01430=-160758,-112853,-114863,36163,82877,78288
C01431=-160760,-113152,-111426,36317,81029,77674
C01432=-159491,-108015,-113138,31549,97627,78488
C01433=-160662,-113202,-114930,31505,96709,77777
C01434=-163626,-124672,-119545,29271,98661,76908
C01435=-164622,-129006,-121133,28240,99357,76613
C01436=-160757,-112482,-116558,30024,102576,77779
C01437=-160755,-111254,-119690,30396,104801,78387
C01438=-139139,-104942,-132434,5076,105021,81413
C01439=-120610,-140892,-128239,-26796,83300,73925
C01440=-124485,-139346,-124335,-26282,80622,73071
C01441=-128794,-174695,-130569,-28116,58521,76693
C01442=-123854,-173705,-127920,-33486,56775,79744
C01443=-127596,-155142,-123084,-28725,56836,77726
C01444=-128095,-155529,-122172,-29132,53686,78388
C01445=-128860,-155984,-126780,-25446,58633,74277
C01446=-138109,-135032,-133743,-8289,74304,51513
C01447=-203654,-125968,-124215,37381,73551,-30645
C01448=-201127,-103516,-110680,20461,62884,-59060
C01449=-201138,-104157,-107983,20829,61019,-59420
C01450=-201193,-104400,-106652,21043,60147,-59612
C01451=-201232,-104446,-106694,21063,60161,-59627
C01452=-200873,-105228,-106882,20926,59802,-59552
C01453=-201116,-104130,-107973,20816,61021,-59411
C01454=-201105,-103488,-110669,20449,62886,-59051
C01455=-198523,-119273,-121454,24683,77158,-64296
C01456=-174403,-100049,-121231,21877,99309,-62114
C01457=-174406,-102879,-118773,21681,96545,-62622
C01458=-172958,-103152,-117900,21399,95556,-62302
C01459=-174224,-104881,-115910,21520,93897,-63036
C01460=-174418,-104205,-117181,21599,94999,-62906
C01461=-174415,-101880,-119808,21752,97619,-62429
C01462=-185776,-93152,-118465,-1785,83350,-67432
C01463=-169060,-142396,-123848,-37084,49654,-60484
C01464=-174230,-113472,-108308,-34615,49911,-64397
C01465=-174247,-112967,-104740,-35556,48304,-63744
C01466=-174471,-112928,-103062,-35946,47380,-63468
C01467=-174489,-112275,-102294,-36008,47261,-63425
C01468=-174590,-112153,-101603,-36140,46922,-63333
C01469=-174396,-113097,-100663,-36857,46141,-62871
C01470=-174330,-114043,-100633,-37190,45762,-62656
C01471=-174129,-122060,-98220,-45554,37107,-60115
C01472=-174246,-112406,-102200,-36228,47262,-63291
C01473=-174229,-113129,-105847,-35265,48804,-63944
C01474=-182962,-136134,-123657,-29797,44727,-67038
C01475=-203654,-125968,-124215,37381,73551,-30645
C01476=-201127,-103516,-110680,20461,62884,-59060
C01477=-201138,-104157,-107983,20829,61019,-59420
C01478=-201193,-104400,-106652,21043,60147,-59612
C01479=-201232,-104446,-106694,21063,60161,-59627
C01480=-200873,-105228,-106882,20926,59802,-59552
C01481=-201116,-104130,-107973,20816,61021,-59411
C01482=-201105,-103488,-110669,20449,62886,-59051
C01483=-198523,-119273,-121454,24683,77158,-64296
C01484=-174403,-100049,-121231,21877,99309,-62114
C01485=-174406,-102879,-118773,21681,96545,-62622
C01486=-172958,-103152,-117900,21399,95556,-62302
C01487=-174224,-104881,-115910,21520,93897,-63036
C01488=-174418,-104205,-117181,21599,94999,-62906
C01489=-174415,-101880,-119808,21752,97619,-62429
C01490=-185776,-93152,-118465,-1785,83350,-67432
C01491=-169060,-142396,-123848,-37084,49654,-60484
C01492=-174230,-113472,-108308,-34615,49911,-64397
C01493=-174247,-112967,-104740,-35556,48304,-63744
C01494=-174471,-112928,-103062,-35946,47380,-63468
C01495=-174489,-112275,-102294,-36008,47261,-63425
C01496=-174590,-112153,-101603,-36140,46922,-63333
C01497=-174396,-113097,-100663,-36857,46141,-62871
C01498=-174330,-114043,-100633,-37190,45762,-62656
C01499=-174129,-122060,-98220,-45554,37107,-60115
C01500=-174246,-112406,-102200,-36228,47262,-63291
C01501=-175798,-117006,-109100,-34199,48210,-64559
C01502=-178617,-124532,-114828,-32467,46840,-65534
C01503=-210827,-121899,-127370,-35396,86436,-76908
C01504=-214505,-124636,-123608,-35577,86411,-76994
C01505=-214521,-124823,-120077,-35640,84542,-76397
C01506=-209595,-138372,-118962,-40572,76618,-76704
C01507=-215572,-134536,-117924,-37557,71164,-81051
C01508=-214545,-124844,-120083,-35636,84527,-76402
C01509=-214528,-124659,-123615,-35573,86395,-76999
C01510=-214596,-124890,-121786,-39550,96156,-78039
C01511=-214607,-124784,-118461,-39383,94595,-77461
C01512=-215336,-122839,-115954,-39308,93846,-77495
C01513=-215216,-123286,-113688,-39218,92622,-76995
C01514=-214785,-119888,-114308,-39371,94481,-77497
C01515=-214619,-124823,-118761,-39395,94718,-77513
C01516=-214540,-124430,-116246,-48349,86426,-68042
C01517=-214499,-123956,-126099,-48385,90728,-70182
C01518=-158797,-145907,-128305,-56145,74291,-56792
C01519=-118138,-117595,-113507,-59219,64127,-52420
C01520=-134091,-119062,-102284,-58108,50235,-52331
C01521=-134095,-117716,-98836,-59129,49460,-51612
C01522=-134657,-117185,-97454,-59366,48806,-51448
C01523=-134083,-121591,-110246,-11584,43366,-62365
C01524=-133895,-121523,-110170,-11744,43379,-62274
C01525=-133843,-121378,-109751,-11603,42967,-62923
C01526=-134088,-120272,-105685,-8075,39028,-71413
C01527=-134097,-120880,-107281,-7954,39689,-71484
C01528=-133538,-122024,-122159,-7272,48238,-71950
C01529=-134045,-120979,-109361,-39707,45136,-55893
C01530=-134048,-117179,-98466,-43015,41514,-53843
C01531=-133905,-117568,-98535,-40781,40764,-54269
C01532=-134181,-118830,-102497,-12918,37668,-61575
C01533=-134198,-119226,-102647,-12934,37556,-61565
C01534=-167359,-106948,-94294,44068,50330,-74802
C01535=-162364,-123197,-107171,35832,43944,-75497
C01536=-134045,-120979,-109361,-39707,45136,-55893
C01537=-132003,-121638,-109572,-41117,45917,-55073
C01538=-131002,-106489,-98392,-41164,47077,-55091
C01539=-131123,-103588,-88252,-50265,40796,-51296
C01540=-163242,-98975,-95762,18008,45953,-74760
C01541=-153405,-104865,-97946,10266,42608,-70493
C01542=-134148,-119761,-102793,-13034,37388,-61506
C01543=-126986,-126229,-93303,56145,28917,-85918
C01544=-131099,-132353,-104040,54087,33374,-85008
C01545=-133651,-114033,-99266,51853,45977,-77066
C01546=-134816,-132236,-131789,-6177,48808,-72548
C01547=-152519,-98596,-126841,-17039,86437,-59409
C01548=-167034,-82548,-116958,-26153,108191,-47353
C01549=-167227,-85698,-113927,-25595,104988,-46679
C01550=-154754,-79329,-105712,-37422,108521,-45283
C01551=-159285,-74428,-103512,-37136,107681,-46815
C01552=-167896,-62467,-97746,-36329,106502,-49789
C01553=-170836,-57718,-95291,-35960,106173,-50801
C01554=-180979,-58723,-101497,-23976,107062,-51805
C01555=-180909,-54943,-104050,-24554,110296,-52487
C01556=-168157,-75412,-102271,-33648,91006,-21456
C01557=-174012,-67106,-91297,-33471,82630,-14810
C01558=-175466,-61382,-85667,-32996,81659,-15067
C01559=-176013,-59150,-83405,-32819,81253,-15153
C01560=-202608,-62025,-89962,4221,78254,-36710
C01561=-159972,-87195,-101610,-14286,75081,-22762
C01562=-154310,-93015,-102157,-19304,70769,-24486
C01563=-154362,-96202,-104591,-19297,70625,-24481
C01564=-154503,-104813,-110762,-19306,69999,-24428
C01565=-155575,-73729,-96860,-32555,86012,-14938
C01566=-157088,-68154,-91284,-32096,84992,-15206
C01567=-157731,-66276,-89193,-31903,84490,-15302
C01568=-176839,-77218,-97385,-7105,75561,-28432
C01569=-165473,-80321,-98709,-11948,76053,-24715
C01570=-199796,-81518,-91231,35244,71315,-57262
C01571=-201423,-82172,-92479,35779,72324,-57601
C01572=-205660,-83542,-95477,37134,74990,-58446
C01573=-150225,-90058,-124320,-20069,81923,-14603
C01574=-88917,-116100,-126028,-29630,66347,39612
C01575=-48102,-114880,-112674,-35477,56596,75725
C01576=-53396,-105773,-101201,-33500,52497,74682
C01577=-53385,-105323,-98106,-34230,51099,75219
C01578=-48465,-101460,-95464,-40425,56724,79171
C01579=-72122,-108844,-98440,461,39847,55622
C01580=-53363,-105522,-99057,-19217,46878,60217
C01581=-53371,-105892,-101942,-18746,48378,59901
C01582=-53322,-113038,-104699,812,43724,42660
C01583=-53318,-112442,-102021,830,42382,42650
C01584=-53317,-112163,-100935,837,41857,42645
C01585=-53253,-112229,-97736,1547,37461,42516
C01586=-53300,-111445,-98358,1568,38246,42506
C01587=-51520,-115460,-104005,-179,39644,43460
C01588=-55761,-139961,-122674,-27476,66843,55729
C01589=-53542,-121644,-113892,-40363,83761,61539
C01590=-53523,-121175,-111327,-40444,82737,61941
C01591=-53533,-120846,-110023,-41635,87424,59647
C01592=-53533,-120798,-109834,-41636,87355,59676
C01593=-53529,-120315,-108043,-41648,86710,59935
C01594=-53536,-120580,-109029,-41640,87063,59791
C01595=-53556,-121151,-111460,-41628,87965,59422
C01596=-52633,-122748,-126719,-40391,89833,59612
C01597=-140119,-108661,-130674,-21165,82789,-25459
C01598=-161125,-123349,-120158,-18581,66270,-46079
C01599=-161135,-123185,-116439,-18891,64175,-45732
C01600=-161140,-122976,-114905,-19018,63381,-45597
C01601=-161216,-123269,-115002,-18998,63277,-45609
C01602=-162856,-121662,-114495,-18189,63396,-46272
C01603=-161212,-123488,-116538,-18871,64068,-45743
C01604=-161202,-123677,-120265,-18562,66156,-46089
C01605=-167124,-146469,-125858,32695,63076,-70922
C01606=-161220,-122264,-110536,44525,64077,-74742
C01607=-161219,-121375,-107584,44985,63095,-75224
C01608=-164956,-113855,-102560,48427,66781,-75111
C01609=-161213,-120936,-106323,43985,60856,-74418
C01610=-161480,-119492,-104017,44742,56174,-74995
C01611=-161477,-119788,-101535,47560,52624,-77093
C01612=-161197,-119682,-102993,46927,53134,-76618
C01613=-161197,-120736,-105876,46275,53998,-76117
C01614=-161177,-121556,-108554,35078,57327,-43050
C01615=-161177,-120932,-106617,35398,56609,-43319
C01616=-152937,-127654,-109782,25136,48983,-42100
C01617=-161176,-119640,-103030,36318,54707,-44163
C01618=-161179,-121241,-107541,34339,64662,-45277
C01619=-161179,-121533,-108462,34233,65010,-45160
C01620=-161180,-122193,-110741,33972,65899,-44866
C01621=-159909,-111206,-128347,-10927,59798,-43136
C01622=-174276,-119239,-128019,9099,73009,32604
C01623=-174287,-122281,-118814,9519,65873,32039
C01624=-174304,-122135,-115653,9666,64029,31878
C01625=-174310,-121974,-114355,9727,63324,31815
C01626=-174277,-122172,-120616,-9764,82080,37769
C01627=-174277,-122177,-120568,-9764,82048,37772
C01628=-174317,-121775,-113110,-33515,107538,43031
C01629=-174312,-121937,-114098,-33622,107981,42892
C01630=-174299,-122214,-116525,-33911,109120,42531
C01631=-174287,-119835,-127268,-36019,115609,40290
C01632=-174287,-120021,-127206,9145,72119,32532
C01633=-174287,-120021,-127206,9145,72119,32532
C01634=-173736,-117333,-114872,9262,65925,32245
C01635=-174960,-111711,-111152,9771,66659,31859
C01636=-176831,-126585,-121826,-8311,79476,36809
C01637=-157010,-133467,-117360,-32643,99223,56368
C01638=-157552,-135759,-118018,-32604,98358,56401
C01639=-154345,-130153,-124672,-33336,105500,55567
C01640=-146682,-141770,-131473,-27794,101884,56245
C01641=-146682,-141770,-131473,-27794,101884,56245
C01642=-146682,-141770,-131473,15257,98468,53705
C01643=-102938,-141770,-131473,49664,98468,53705
C01644=-102938,-145417,-131473,49512,65454,53705
C01645=-103656,-129714,-109721,51674,62395,51470
C01646=-102995,-138917,-102303,63406,51064,43511
C01647=-104839,-135559,-111699,50177,75701,60454
C01648=-99828,-171084,-120161,53403,64595,56658
C01649=-110163,-126067,-103455,56717,91063,66073
C01650=-116435,-131456,-112749,56730,96510,65994
C01651=-116383,-133294,-113279,56655,96128,65766
C01652=-84454,-125099,-129012,35107,90636,33075
C01653=-15972,-110889,-128286,-10965,59905,-43045
C01654=-15972,-110889,-128286,-10965,59905,-43045
C01655=-53465,-86935,-89811,-40465,79071,68727
C01656=-108812,15435,-43443,-8262,104585,64007
C01657=-120685,104729,62045,12414,91835,74489
C01658=-120504,102152,62779,12366,90072,74374
C01659=-120431,101212,63194,12350,89339,74325
C01660=-120431,101002,64582,12347,88398,74232
C01661=-120431,101212,63194,12350,89339,74325
C01662=-121076,107244,72775,12456,86702,73844
C01663=-120665,102968,67176,12385,87860,74099
C01664=-121076,107244,72775,12456,86702,73844
C01665=-121323,110426,71256,12493,89251,74016
C01666=-131278,69881,50181,9127,63188,62805
C01667=-131485,74883,60411,9547,59533,62414
C01668=-131548,76399,63510,9674,58426,62296
C01669=-131548,76704,64506,9721,57977,62255
C01670=-131183,71204,57206,9397,59578,62541
C01671=-131068,71487,58412,9405,58972,62536
C01672=-131266,74091,61533,9552,58423,62408
C01673=-131382,69379,53589,9372,60872,62574
C01674=-130781,63634,40058,8705,66118,63219
C01675=-132526,40318,17232,-3897,63337,79864
C01676=-132770,43850,25861,-3900,59836,79894
C01677=-132775,45020,27808,-3921,59239,79913
C01678=-132775,45119,28557,-3937,58830,79928
C01679=-131974,40901,23457,-4303,59840,80201
C01680=-131974,41007,24367,-4325,59336,80221
C01681=-132343,43569,27070,-4148,58978,80090
C01682=-132425,41720,24361,-4076,59689,80031
C01683=-131916,36045,14544,-4216,62827,80109
C01684=-154350,3292,-38754,752,86522,75713
C01685=-181553,89062,52820,1715,95022,75090
C01686=-181735,85640,53357,1725,92938,75001
C01687=-181765,85113,53499,1727,92580,74986
C01688=-181767,85098,55139,1725,91564,74972
C01689=-181765,85113,53499,1727,92580,74986
C01690=-181351,93067,65191,1686,89465,75083
C01691=-181572,88775,59771,1706,90599,75024
C01692=-181351,93067,65191,1686,89465,75083
C01693=-181147,96755,64289,1671,91909,75184
C01694=-159394,22511,-602,-1012,64107,82504
C01695=-159231,25736,7387,-1125,60850,82595
C01696=-159081,26911,9255,-1209,60307,82658
C01697=-159081,26976,10155,-1214,59786,82663
C01698=-159081,26911,9255,-1209,60307,82658
C01699=-159295,23244,6238,-1098,60277,82577
C01700=-159295,23278,6733,-1101,59990,82580
C01701=-159347,25129,8513,-1077,59844,82563
C01702=-159295,23278,6733,-1101,59990,82580
C01703=-159427,17860,-3265,-1001,63356,82499
C01704=-180998,44453,11386,9428,69103,75000
C01705=-180806,46143,18147,9552,65832,74803
C01706=-180780,46418,19112,9573,65382,74775
C01707=-180783,46335,20682,9650,64387,74690
C01708=-180780,46418,19112,9573,65382,74775
C01709=-181199,40700,14756,9793,65178,74604
C01710=-180944,43672,17889,9700,64752,74662
C01711=-181199,40700,14756,9793,65178,74604
C01712=-181427,38720,7071,9647,68865,74830
C01713=-152316,-9212,-39627,-4041,74028,47424
C01714=-97675,-116344,-75406,-30929,43249,-3453
C01715=-144147,-96317,-43020,16665,22045,18189
C01716=-130185,-5552,7433,-2044,36537,82607
C01717=-148170,9866,-4864,-2727,74191,81047
C01718=-160677,16615,-6140,-3325,93789,80088
C01719=-160892,14618,-3978,-3294,91428,80078
C01720=-160979,13901,-3035,-3283,90476,80074
C01721=-160981,13982,-1301,-3281,89453,80100
C01722=-160979,13901,-3035,-3283,90476,80074
C01723=-160903,19705,2788,-3289,89879,80114
C01724=-160903,19733,3315,-3289,89569,80123
C01725=-160898,16854,1424,-3289,89254,80133
C01726=-160903,19794,4169,-3288,89076,80136
C01727=-160610,22295,943,-3323,92353,80148
C01728=-159769,-26352,-42847,7626,75430,42908
C01729=-160661,-23608,-37245,8003,73495,42476
C01730=-160801,-19429,-32426,8083,72699,42375
C01731=-160801,-19408,-31304,8110,72027,42329
C01732=-161009,-22449,-34949,8156,72720,42303
C01733=-161249,-23550,-34138,8284,71688,42148
C01734=-161035,-21507,-32672,8205,71812,42231
C01735=-161249,-23550,-34138,8284,71688,42148
C01736=-159612,-30937,-44211,7622,73912,42867
C01737=-144117,-44081,-61004,-17211,89666,8724
C01738=-145648,-40124,-55468,-16926,88039,8426
C01739=-146237,-38515,-53215,-16819,87384,8313
C01740=-146244,-38444,-53170,-16818,87391,8310
C01741=-146245,-38577,-51594,-16825,86395,8446
C01742=-146244,-38444,-53170,-16818,87391,8310
C01743=-146240,-38608,-52193,-16823,86734,8401
C01744=-146535,-35573,-50236,-16765,87015,8261
C01745=-146268,-38521,-51765,-16819,86519,8421
C01746=-147801,-39090,-52130,-16535,86146,7942
C01747=-146268,-38521,-51765,-16819,86519,8421
C01748=-144117,-44081,-61004,-17211,89666,8724
C01749=-145162,-56828,-95851,-3587,97052,36303
C01750=-147136,-55674,-91646,-3015,94990,35768
C01751=-150906,-56103,-90461,-1950,93937,34650
C01752=-150909,-57277,-89363,-1945,92659,34669
C01753=-150906,-56103,-90461,-1950,93937,34650
C01754=-147900,-55107,-89916,-2796,94193,35556
C01755=-147871,-56692,-89008,-2798,92822,35595
C01756=-149697,-57326,-89351,-2285,92656,35040
C01757=-147871,-56692,-89008,-2798,92822,35595
C01758=-149264,-52275,-86592,-2410,93564,35155
C01759=-149536,-48545,-84471,-2336,94168,35061
C01760=-149264,-52275,-86592,-2410,93564,35155
C01761=-145162,-56828,-95851,-3587,97052,36303
C01762=-148725,-41791,-46801,-46253,72923,-63254
C01763=-150766,-40622,-42529,-46203,70442,-63063
C01764=-151577,-40068,-40761,-46203,69457,-62988
C01765=-152585,-23504,-29643,-45527,70124,-63820
C01766=-151861,-23991,-31407,-45521,71087,-63922
C01767=-150038,-24992,-35653,-45558,73508,-64179
C01768=-157424,-58492,-62688,-32217,54755,-56547
C01769=-158288,-54308,-56839,-32290,53193,-56420
C01770=-158489,-51803,-54002,-32356,52725,-56354
C01771=-162920,-52118,-54243,-29783,51091,-57961
C01772=-162018,-54402,-56899,-30142,51809,-57760
C01773=-161259,-58664,-62788,-30049,53328,-57890
C01774=-162071,-38381,-52824,-22779,71448,-67723
C01775=-163630,41,-22976,-9730,99876,-85306
C01776=-164211,-2681,-21394,-9632,97468,-85315
C01777=-164465,-2984,-20111,-9597,96504,-85326
C01778=-167232,-2580,-19786,-9490,96192,-86245
C01779=-166888,-2331,-21114,-9528,97164,-86203
C01780=-166273,343,-22730,-9627,99573,-86181
C01781=-147061,-19099,-23009,-3757,61390,-3418
C01782=-130185,-5552,7433,-2044,36537,20417
C01783=-144147,-96317,-43020,16665,22045,18189
C01784=-97675,-116344,-75406,-30929,43249,-3453
C01785=-152316,-9212,-39627,-4041,74028,-36586
C01786=-151393,-4993,-15312,-4384,44467,-75506
C01787=-149831,-2435,-10935,-5835,43191,-74682
C01788=-153598,-2863,-5088,4597,34036,-78104
C01789=-153144,-5743,-2041,16094,25401,-81582
C01790=-154914,-1885,-10222,12324,42496,-79899
C01791=-154718,-4280,-13376,11999,43163,-79709
C01792=-167718,15574,1984,-24206,55458,-53961
C01793=-167855,19598,9384,-24857,53146,-53442
C01794=-167909,21312,12472,-25150,52202,-53220
C01795=-169559,21751,12884,-24222,51683,-53852
C01796=-169779,21817,12946,-24097,51615,-53936
C01797=-170327,21990,13109,-23783,51447,-54148
C01798=-170290,20267,10006,-23488,52399,-54367
C01799=-170195,16223,2573,-22831,54729,-54878
C01800=-178256,99378,67031,-19051,88552,-69176
C01801=-178526,97657,68868,-19024,86580,-68963
C01802=-178635,97078,69748,-19021,85760,-68874
C01803=-179853,98823,71988,-18874,85023,-69192
C01804=-179980,99017,72237,-18859,84943,-69225
C01805=-180384,99643,73043,-18810,84684,-69328
C01806=-180272,100173,72105,-18809,85516,-69417
C01807=-179996,101790,70145,-18825,87512,-69628
C01808=-171488,21123,-18735,-439,89529,-9365
C01809=-148539,8283,-18518,11481,74800,46031
C01810=-133884,78471,30098,11624,77529,65496
C01811=-133939,79564,34318,11736,75541,65288
C01812=-133726,80326,36877,11703,74352,65242
C01813=-129986,86296,44341,10172,72375,66337
C01814=-130560,84597,41197,10369,73487,66234
C01815=-130480,83524,36335,10225,75880,66464
C01816=-133789,96970,48697,23463,95575,62558
C01817=-133554,94997,50328,23328,93653,62262
C01818=-133996,90156,45840,23419,94027,62179
C01819=-133380,91261,47236,23299,93592,62310
C01820=-133261,94504,51359,23246,92757,62189
C01821=-128474,99178,56254,18479,90935,62982
C01822=-126544,95607,50814,14280,92008,63224
C01823=-126033,96144,51503,14181,91777,63369
C01824=-125984,92855,44553,14229,94278,63672
C01825=-118409,86943,34254,-498,98079,29639
C01826=-113225,75702,29820,-12477,90617,28537
C01827=-112952,75485,30802,-12536,89960,28691
C01828=-117762,67578,21374,-3134,88425,17539
C01829=-120996,68894,22851,4133,88343,9509
C01830=-120986,83403,30534,4203,100743,9917
C01831=-131138,87625,41047,12528,91017,-11277
C01832=-131518,88313,46232,13974,85364,-12988
C01833=-131574,88042,47103,13998,84717,-13081
C01834=-131699,87452,47047,14037,84474,-13150
C01835=-127523,76387,33616,3918,83280,-1876
C01836=-130224,83461,42270,11062,83726,-9611
C01837=-130883,82631,32190,11215,89482,-9310
C01838=-138903,29280,-14444,28707,91021,50587
C01839=-152753,-113498,-70464,41238,43505,17390
C01840=-199062,-57325,-47228,38260,64183,4080
C01841=-144700,-70309,-53328,-41384,55522,-26317
C01842=-159027,-8981,-29340,-14833,99808,-55594
C01843=-158734,-10357,-26337,-14717,97386,-55198
C01844=-158565,-10606,-24902,-14680,96435,-55024
C01845=-156379,-10444,-24769,-14732,96828,-54309
C01846=-156533,-10130,-26155,-14772,97783,-54479
C01847=-156840,-8773,-29171,-14894,100200,-54881
C01848=-162486,-26662,-42491,-16083,70936,-60571
C01849=-162478,-24897,-37244,-16311,68704,-60258
C01850=-161179,-32593,-36996,-20221,58130,-58095
C01851=-158572,-32392,-36861,-21515,58809,-57144
C01852=-159367,-24765,-36916,-18592,69259,-59149
C01853=-159276,-26541,-42171,-18380,71485,-59471
C01854=-144700,-70309,-53328,-41384,55522,-26317
C01855=-199062,-57325,-47228,38260,64183,4080
C01856=-152753,-113498,-70464,41238,43505,17390
C01857=-138903,29280,-14444,28707,91021,50587
C01858=-134460,43790,22046,6339,61230,73811
C01859=-133863,45767,26803,6146,59285,73930
C01860=-134087,48465,31540,6362,57781,73758
C01861=-130025,54134,37725,4242,56630,75317
C01862=-129992,52392,35365,4200,57178,75352
C01863=-129939,49644,28351,4047,60072,75482
C01864=-131463,16549,-4479,-10803,54184,75739
C01865=-132193,19578,1957,-10644,51724,75694
C01866=-132626,21348,4069,-10405,51283,75555
C01867=-134889,19383,2337,-8835,51077,74604
C01868=-134234,16346,-1785,-9163,52111,74787
C01869=-134362,13693,-7099,-8856,53981,74568
C01870=-136755,-2244,-27091,-2141,60146,66966
C01871=-152753,-113498,-70464,41238,43505,17390
C01872=-199062,-57325,-47228,38260,64183,4080
C01873=-144700,-70309,-53328,-41384,55522,-26317
C01874=-155243,-37029,-47289,-14287,81392,-50093
C01875=-162013,-14853,-33688,2862,92831,-64763
C01876=-161094,-16180,-30749,2749,90312,-64514
C01877=-160723,-16617,-29501,2705,89308,-64411
C01878=-157149,-16390,-29322,2290,89205,-63218
C01879=-157529,-15990,-30598,2335,90205,-63327
C01880=-158470,-14757,-33607,2451,92716,-63592
C01881=-164755,-27863,-42732,4142,59506,-66566
C01882=-163775,-25128,-37158,3650,57439,-66261
C01883=-162063,-21722,-33626,2650,56947,-65603
C01884=-158969,-21729,-33662,803,56902,-64386
C01885=-159524,-25179,-37184,1127,57304,-64599
C01886=-160428,-28024,-42833,1630,59333,-64922
C01887=-144700,-70309,-53328,-41384,55522,-26317
C01888=-199062,-57325,-47228,38260,64183,4080
C01889=-152753,-113498,-70464,41238,43505,17390
C01890=-177120,62510,20627,9539,95868,-53949
C01891=-182918,102274,70865,2025,89904,-72285
C01892=-182573,99881,71746,1990,88125,-72198
C01893=-182434,99026,72237,1977,87381,-72163
C01894=-177980,92594,64030,1535,89029,-70642
C01895=-178132,93443,63515,1551,89785,-70684
C01896=-178509,95798,62536,1591,91604,-70787
C01897=-170148,25411,11260,-10861,54110,-56839
C01898=-169779,29504,18940,-11463,51585,-56403
C01899=-169678,31092,21995,-11696,50557,-56237
C01900=-164974,29903,20823,-14564,51428,-54281
C01901=-165316,28440,17904,-14160,52381,-54569
C01902=-165615,24318,10218,-13532,54869,-55036
C01903=-177120,62510,20627,9539,95868,-53949
C01904=-152753,-113498,-70464,41238,43505,17390
C01905=-199062,-57325,-47228,38260,64183,4080
C01906=-144700,-70309,-53328,-41384,55522,-26317
C01907=-142540,-54200,-62960,-20837,71495,-76935
C01908=-143745,-53250,-58469,-20670,69060,-76947
C01909=-143907,-52449,-56432,-20721,68229,-76859
C01910=-146015,-19661,-41212,-16744,94255,-78829
C01911=-145325,-27004,-46307,-16815,93781,-78527
C01912=-145058,-29561,-48130,-16841,93649,-78418
C01913=-144903,-28900,-49357,-16896,94730,-78514
C01914=-144163,-26309,-51550,-17103,97446,-78641
C01915=-174273,-50790,-66274,-423,45257,-81721
C01916=-174293,-46300,-60313,-415,43895,-81724
C01917=-174300,-44502,-57900,-412,43334,-81724
C01918=-174308,-44682,-54936,-420,41418,-81719
C01919=-174300,-46542,-57382,-423,41967,-81718
C01920=-174281,-51187,-63424,-430,43299,-81715
C01921=-170286,-21589,-54734,-4189,80944,-76248
C01922=-174005,35790,2399,-5860,112639,-83034
C01923=-174229,31517,1683,-5803,110877,-83024
C01924=-174320,29862,1474,-5782,110152,-83021
C01925=-174151,30232,3489,-5706,109139,-82910
C01926=-174234,31116,4346,-5726,109041,-82935
C01927=-174010,35219,4888,-5776,110822,-82944
C01928=-165073,-12180,-39998,-12766,95090,-81399
C01929=-146454,-66354,-59123,-37370,62542,-80053
C01930=-148014,-113391,-77231,-42747,49474,-76607
C01931=-120872,-104982,-67229,-50399,61266,-16237
C01932=-12667,-135547,-130714,31270,45596,0
BC00000=78393,670967,1075175
BC00001=177059,727519,1002542
BC00002=78393,913126,1075175
BC00003=70793,903989,1075175
BC00004=70793,903989,1075175
BC00005=70793,903989,1075175
BC00006=70793,903989,1075175
BC00007=70793,903989,1075175
BC00008=70793,903989,1075175
BC00009=70793,903989,1075175
BC00010=70793,903989,1075175
BC00011=70793,903989,1075175
BC00012=103901,897249,1075175
BC00013=103901,897249,1075175
BC00014=103901,897249,1075175
BC00015=103901,897249,1075175
BC00016=103901,897249,1075175
BC00017=103901,897249,1075175
BC00018=103901,897249,1075175
BC00019=103901,897249,1075175
BC00020=89915,910531,1075175
BC00021=89915,910531,1075175
BC00022=89916,910530,1075174
BC00023=89916,910530,1075174
BC00024=89916,910530,1075174
BC00025=89916,910530,1075174
BC00026=89916,910530,1075174
BC00027=89916,910530,1075174
BC00028=89916,910530,1075174
BC00029=89915,910531,1075175
BC00030=89915,910531,1075175
BC00031=89915,910531,1075175
BC00032=89915,910531,1075175
BC00033=89915,910531,1075175
BC00034=89915,910531,1075175
BC00035=89915,910531,1075175
BC00036=27368,899646,1075175
BC00037=27368,899646,1075175
BC00038=27368,899646,1075175
BC00039=27368,899646,1075175
BC00040=27368,899646,1075175
BC00041=27368,899646,1075175
BC00042=27368,899646,1075175
BC00043=27368,899646,1075175
BC00044=160753,772187,1075175
BC00045=160753,772187,1075175
BC00046=160753,772187,1075175
BC00047=160753,772187,1075175
BC00048=160753,772187,1075175
BC00049=160753,772187,1075175
BC00050=160753,772187,1075175
BC00051=160753,772187,1075175
BC00052=160753,772187,1075175
BC00053=160753,772187,1075175
BC00054=160753,772187,1075175
BC00055=160753,772187,1075175
BC00056=123402,765716,1075175
BC00057=123402,765716,1075175
BC00058=123402,765716,1075175
BC00059=123402,765716,1075175
BC00060=123402,765716,1075175
BC00061=123402,765716,1075175
BC00062=123402,765716,1075175
BC00063=123402,765716,1075175
BC00064=123402,765716,1075175
BC00065=123402,765716,1075175
BC00066=123402,765716,1075175
BC00067=129464,768278,1075175
BC00068=151149,777443,1075175
BC00069=169689,785624,1075175
BC00070=169689,785624,1075175
BC00071=169689,785624,1075175
BC00072=169689,785624,1075175
BC00073=169689,785624,1075175
BC00074=169689,785624,1075175
BC00075=169689,785624,1075175
BC00076=169689,785624,1075175
BC00077=169689,785624,1075175
BC00078=169689,785624,1075175
BC00079=169689,785624,1075175
BC00080=169689,785624,1075175
BC00081=169689,785624,1075175
BC00082=120114,813651,1075175
BC00083=120114,813651,1075175
BC00084=120114,813651,1075175
BC00085=120114,813651,1075175
BC00086=120114,813651,1075175
BC00087=120114,813651,1075175
BC00088=120114,813651,1075175
BC00089=120114,813651,1075175
BC00090=120114,813651,1075175
BC00091=120114,813651,1075175
BC00092=120114,813651,1075175
BC00093=120114,813651,1075175
BC00094=120114,813651,1075175
BC00095=141881,838168,1075175
BC00096=141881,838168,1075175
BC00097=141881,838168,1075175
BC00098=141881,838168,1075175
BC00099=141881,838168,1075175
BC00100=141881,838168,1075175
BC00101=141881,838168,1075175
BC00102=141881,838168,1075175
BC00103=141881,838168,1075175
BC00104=141881,838168,1075175
BC00105=141881,838168,1075175
BC00106=141881,838168,1075175
BC00107=141881,838168,1075175
BC00108=69874,805894,1075175
BC00109=70019,750208,1075175
BC00110=70019,750208,1075175
BC00111=70019,750208,1075175
BC00112=70019,750208,1075175
BC00113=70019,750208,1075175
BC00114=70019,750208,1075175
BC00115=70019,750208,1075175
BC00116=70019,750208,1075175
BC00117=70019,750208,1075175
BC00118=70019,750208,1075175
BC00119=70019,750208,1075175
BC00120=70019,750208,1075175
BC00121=70019,750208,1075175
BC00122=70018,750208,1075172
BC00123=70018,750208,1075172
BC00124=70018,750208,1075172
BC00125=70018,750208,1075172
BC00126=70018,750208,1075172
BC00127=70018,750208,1075172
BC00128=70018,750208,1075172
BC00129=70018,750208,1075172
BC00130=110204,822960,1075174
BC00131=128430,855958,1075175
BC00132=125005,945340,1075175
BC00133=125005,945340,1075175
BC00134=125005,945340,1075174
BC00135=125005,945340,1075174
BC00136=125005,945340,1075174
BC00137=125005,945340,1075174
BC00138=125005,945340,1075174
BC00139=125005,945340,1075174
BC00140=125005,945340,1075174
BC00141=125005,945340,1075174
BC00142=125005,945340,1075175
BC00143=143574,943463,1075175
BC00144=143574,943463,1075175
BC00145=143574,943463,1075175
BC00146=143574,943463,1075175
BC00147=143574,943463,1075175
BC00148=143574,943463,1075175
BC00149=143574,943463,1075175
BC00150=177748,940008,1075175
BC00151=177748,940008,1075175
BC00152=177748,940008,1075175
BC00153=177748,940008,1075175
BC00154=177748,940008,1075175
BC00155=177748,940008,1075175
BC00156=177748,940008,1075175
BC00157=177748,940008,1075175
BC00158=177748,940008,1075175
BC00159=177748,940008,1075175
BC00160=177748,940008,1075175
BC00161=177748,940008,1075175
BC00162=225975,953000,1075175
BC00163=225975,953000,1075175
BC00164=225975,953000,1075175
BC00165=225975,953000,1075175
BC00166=225975,953000,1075175
BC00167=225975,953000,1075175
BC00168=225975,953000,1075175
BC00169=183095,975695,1075175
